			TT_01_01													:= m01_rs1_r1._01_TT_01,
			TT_01_01_offset												:= m01_rs1_r1.cart01_front_temp_offset,
			TT_01_01_error												:= m01_rs1_r1._01_TT_01_Error,
			TT_01_03													:= m01_rs1_r1._01_TT_03,               
			TT_01_03_offset												:= m01_rs1_r1.cart01_front_temp_offset,
			TT_01_03_error												:= m01_rs1_r1._01_TT_03_Error,         
			TT_02_01													:= m01_rs1_r1._02_TT_01,               
			TT_02_01_offset												:= m01_rs1_r1.cart02_front_temp_offset,
			TT_02_01_error												:= m01_rs1_r1._02_TT_01_Error,         
			TT_02_03													:= m01_rs1_r1._02_TT_03,               
			TT_02_03_offset												:= m01_rs1_r1.cart02_front_temp_offset,
			TT_02_03_error												:= m01_rs1_r1._02_TT_03_Error,         
			TT_03_01													:= m01_rs1_r1._03_TT_01,               
			TT_03_01_offset												:= m01_rs1_r1.cart03_front_temp_offset,
			TT_03_01_error												:= m01_rs1_r1._03_TT_01_Error,         
			TT_03_03													:= m01_rs1_r1._03_TT_03,               
			TT_03_03_offset												:= m01_rs1_r1.cart03_front_temp_offset,
			TT_03_03_error												:= m01_rs1_r1._03_TT_03_Error,         
			TT_04_01													:= m01_rs1_r1._04_TT_01,               
			TT_04_01_offset												:= m01_rs1_r1.cart04_front_temp_offset,
			TT_04_01_error												:= m01_rs1_r1._04_TT_01_Error,         
			TT_04_03													:= m01_rs1_r1._04_TT_03,               
			TT_04_03_offset												:= m01_rs1_r1.cart04_front_temp_offset,
			TT_04_03_error												:= m01_rs1_r1._04_TT_03_Error,         
			TT_05_01													:= m01_rs1_r1._05_TT_01,               
			TT_05_01_offset												:= m01_rs1_r1.cart05_front_temp_offset,
			TT_05_01_error												:= m01_rs1_r1._05_TT_01_Error,         
			TT_05_03													:= m01_rs1_r1._05_TT_03,               
			TT_05_03_offset												:= m01_rs1_r1.cart05_front_temp_offset,
			TT_05_03_error												:= m01_rs1_r1._05_TT_03_Error,         
			TT_06_01													:= m01_rs1_r1._06_TT_01,               
			TT_06_01_offset												:= m01_rs1_r1.cart06_front_temp_offset,
			TT_06_01_error												:= m01_rs1_r1._06_TT_01_Error,         
			TT_06_03													:= m01_rs1_r1._06_TT_03,               
			TT_06_03_offset												:= m01_rs1_r1.cart06_front_temp_offset,
			TT_06_03_error												:= m01_rs1_r1._06_TT_03_Error,         
			TT_07_01													:= m01_rs1_r1._07_TT_01,               
			TT_07_01_offset												:= m01_rs1_r1.cart07_front_temp_offset,
			TT_07_01_error												:= m01_rs1_r1._07_TT_01_Error,         
			TT_07_03													:= m01_rs1_r1._07_TT_03,               
			TT_07_03_offset												:= m01_rs1_r1.cart07_front_temp_offset,
			TT_07_03_error												:= m01_rs1_r1._07_TT_03_Error,         
			TT_08_01													:= m01_rs1_r1._08_TT_01,               
			TT_08_01_offset												:= m01_rs1_r1.cart08_front_temp_offset,
			TT_08_01_error												:= m01_rs1_r1._08_TT_01_Error,         
			TT_08_03													:= m01_rs1_r1._08_TT_03,               
			TT_08_03_offset												:= m01_rs1_r1.cart08_front_temp_offset,
			TT_08_03_error												:= m01_rs1_r1._08_TT_03_Error,         
			TT_09_01													:= m01_rs1_r1._09_TT_01,               
			TT_09_01_offset												:= m01_rs1_r1.cart09_front_temp_offset,
			TT_09_01_error												:= m01_rs1_r1._09_TT_01_Error,         
			TT_09_03													:= m01_rs1_r1._09_TT_03,               
			TT_09_03_offset												:= m01_rs1_r1.cart09_front_temp_offset,
			TT_09_03_error												:= m01_rs1_r1._09_TT_03_Error,         
			TT_10_01													:= m01_rs1_r1._10_TT_01,               
			TT_10_01_offset												:= m01_rs1_r1.cart10_front_temp_offset,
			TT_10_01_error												:= m01_rs1_r1._10_TT_01_Error,         
			TT_10_03													:= m01_rs1_r1._10_TT_03,               
			TT_10_03_offset												:= m01_rs1_r1.cart10_front_temp_offset,
			TT_10_03_error												:= m01_rs1_r1._10_TT_03_Error,         
			TT_11_01													:= m01_rs1_r1._11_TT_01,               
			TT_11_01_offset												:= m01_rs1_r1.cart11_front_temp_offset,
			TT_11_01_error												:= m01_rs1_r1._11_TT_01_Error,         
			TT_11_03													:= m01_rs1_r1._11_TT_03,               
			TT_11_03_offset												:= m01_rs1_r1.cart11_front_temp_offset,
			TT_11_03_error												:= m01_rs1_r1._11_TT_03_Error,         
			TT_12_01													:= m01_rs1_r1._12_TT_01,               
			TT_12_01_offset												:= m01_rs1_r1.cart12_front_temp_offset,
			TT_12_01_error												:= m01_rs1_r1._12_TT_01_Error,         
			TT_12_03													:= m01_rs1_r1._12_TT_03,               
			TT_12_03_offset												:= m01_rs1_r1.cart12_front_temp_offset,
			TT_12_03_error												:= m01_rs1_r1._12_TT_03_Error,
			
			cart01_front_temp											=> m01_rs1_r1.cart01_front_temp,						
			cart01_front_temp_error 									=> m01_rs1_r1.cart01_front_temp_error,
			cart01_back_temp											=> m01_rs1_r1.cart01_back_temp,
			cart01_back_temp_error 										=> m01_rs1_r1.cart01_back_temp_error,
			cart02_front_temp											=> m01_rs1_r1.cart02_front_temp,						
			cart02_front_temp_error 									=> m01_rs1_r1.cart02_front_temp_error,
			cart02_back_temp											=> m01_rs1_r1.cart02_back_temp,
			cart02_back_temp_error 										=> m01_rs1_r1.cart02_back_temp_error,
			cart03_front_temp											=> m01_rs1_r1.cart03_front_temp,						
			cart03_front_temp_error 									=> m01_rs1_r1.cart03_front_temp_error,
			cart03_back_temp											=> m01_rs1_r1.cart03_back_temp,
			cart03_back_temp_error 										=> m01_rs1_r1.cart03_back_temp_error,
			cart04_front_temp											=> m01_rs1_r1.cart04_front_temp,						
			cart04_front_temp_error 									=> m01_rs1_r1.cart04_front_temp_error,
			cart04_back_temp											=> m01_rs1_r1.cart04_back_temp,
			cart04_back_temp_error 										=> m01_rs1_r1.cart04_back_temp_error,
			cart05_front_temp											=> m01_rs1_r1.cart05_front_temp,						
			cart05_front_temp_error 									=> m01_rs1_r1.cart05_front_temp_error,
			cart05_back_temp											=> m01_rs1_r1.cart05_back_temp,
			cart05_back_temp_error 										=> m01_rs1_r1.cart05_back_temp_error,
			cart06_front_temp											=> m01_rs1_r1.cart06_front_temp,						
			cart06_front_temp_error 									=> m01_rs1_r1.cart06_front_temp_error,
			cart06_back_temp											=> m01_rs1_r1.cart06_back_temp,
			cart06_back_temp_error 										=> m01_rs1_r1.cart06_back_temp_error,
			cart07_front_temp											=> m01_rs1_r1.cart07_front_temp,						
			cart07_front_temp_error 									=> m01_rs1_r1.cart07_front_temp_error,
			cart07_back_temp											=> m01_rs1_r1.cart07_back_temp,
			cart07_back_temp_error 										=> m01_rs1_r1.cart07_back_temp_error,
			cart08_front_temp											=> m01_rs1_r1.cart08_front_temp,						
			cart08_front_temp_error 									=> m01_rs1_r1.cart08_front_temp_error,
			cart08_back_temp											=> m01_rs1_r1.cart08_back_temp,
			cart08_back_temp_error 										=> m01_rs1_r1.cart08_back_temp_error,
			cart09_front_temp											=> m01_rs1_r1.cart09_front_temp,						
			cart09_front_temp_error 									=> m01_rs1_r1.cart09_front_temp_error,
			cart09_back_temp											=> m01_rs1_r1.cart09_back_temp,
			cart09_back_temp_error 										=> m01_rs1_r1.cart09_back_temp_error,
			cart10_front_temp											=> m01_rs1_r1.cart10_front_temp,						
			cart10_front_temp_error 									=> m01_rs1_r1.cart10_front_temp_error,
			cart10_back_temp											=> m01_rs1_r1.cart10_back_temp,
			cart10_back_temp_error 										=> m01_rs1_r1.cart10_back_temp_error,
			cart11_front_temp											=> m01_rs1_r1.cart11_front_temp,						
			cart11_front_temp_error 									=> m01_rs1_r1.cart11_front_temp_error,
			cart11_back_temp											=> m01_rs1_r1.cart11_back_temp,
			cart11_back_temp_error 										=> m01_rs1_r1.cart11_back_temp_error,
			cart12_front_temp											=> m01_rs1_r1.cart12_front_temp,						
			cart12_front_temp_error 									=> m01_rs1_r1.cart12_front_temp_error,
			cart12_back_temp											=> m01_rs1_r1.cart12_back_temp,
			cart12_back_temp_error 										=> m01_rs1_r1.cart12_back_temp_error,
			         
		                                                        
			inlet_co2_pump												:= m01_rs1_r1.inlet_co2_pump,
			AT_01_pump													=> m01_rs1_r1.AT_01_pump,
			inlet_co2_pump_cmd_status									=> m01_rs1_r1.inlet_co2_pump_cmd_status,
			inlet_co2_sol												:= m01_rs1_r1.inlet_co2_sol,
			AT_01_sol													=> m01_rs1_r1.AT_01_sol,
			inlet_co2_sol_cmd_status									=> m01_rs1_r1.inlet_co2_sol_cmd_status,
			outlet_co2_pump												:= m01_rs1_r1.outlet_co2_pump,
			AT_03_pump													=> m01_rs1_r1.AT_03_pump,
			outlet_co2_pump_cmd_status									=> m01_rs1_r1.outlet_co2_pump_cmd_status,
			outlet_co2_sol												:= m01_rs1_r1.outlet_co2_sol,
			AT_03_sol													=> m01_rs1_r1.AT_03_sol,
			outlet_co2_sol_cmd_status									=> m01_rs1_r1.outlet_co2_sol_cmd_status,
			repres_valve												:= m01_rs1_r1.repres_valve,
			XV_02														=> m01_rs1_r1.XV_02,
			repres_valve_open_cmd_status								=> m01_rs1_r1.repres_valve_open_cmd_status,
			repres_valve_open											:= m01_rs1_r1.repres_valve_open,
			repres_valve_closed											:= m01_rs1_r1.repres_valve_closed,
    	                                                        
			fan_vfd_control												=> m01_rs1_r1.fan_vfd_control,  		
			fan_vfd_target_vel	 		                                => m01_rs1_r1.fan_vfd_target_vel, 
			fan_vfd_enabled	 		                                    => m01_rs1_r1.fan_vfd_enabled, 
			fan_vfd_error		                                        => m01_rs1_r1.fan_vfd_error,
			fan_vfd_output												=> m01_rs1_r1.fan_vfd_output,
			fan_vfd_reset												:= m01_rs1_r1.fan_vfd_reset,
			fan_vfd_enable												:= m01_rs1_r1.fan_vfd_enable,
			fan_vfd_ecat_state											:= m01_rs1_r1.fan_vfd_ecat_state,
			fan_vfd_status												:= m01_rs1_r1.fan_vfd_status,
			fan_vfd														:= m01_rs1_r1.fan_vfd,
			fan_vfd_velocity											:= m01_rs1_r1.fan_vfd_velocity,
			fan_vfd_current												:= m01_rs1_r1.fan_vfd_current,
			fan_vfd_current_amps										=> m01_rs1_r1.fan_vfd_output_current,
			fan_vfd_temp												:= m01_rs1_r1.fan_vfd_temp,
			fan_vfd_temp_degC											=> m01_rs1_r1.fan_vfd_temperature,
			                                                    
			inlet_door_clamps_extend									:= m01_rs1_r1.inlet_door_clamps_extend,
			outlet_door_clamps_extend									:= m01_rs1_r1.outlet_door_clamps_extend,
			inlet_door_clamps_retract									:= m01_rs1_r1.inlet_door_clamps_retract,
			outlet_door_clamps_retract									:= m01_rs1_r1.outlet_door_clamps_retract,
			                                                    
			extend_clamps												:= extend_clamps,
			retract_clamps												:= retract_clamps,
			                                                    
			inlet_door_left_clamps_extend								=> m01_rs1_r1.XV_01_Left_Extend_Solenoid_Valve,
			inlet_door_right_clamps_extend								=> m01_rs1_r1.XV_01_Right_Extend_Solenoid_Valve,
			outlet_door_left_clamps_extend								=> m01_rs1_r1.XV_03_Left_Extend_Solenoid_Valve,
			outlet_door_right_clamps_extend								=> m01_rs1_r1.XV_03_Right_Extend_Solenoid_Valve,
			inlet_door_left_clamps_retract								=> m01_rs1_r1.XV_01_Left_Retract_Solenoid_Valve,
			inlet_door_right_clamps_retract								=> m01_rs1_r1.XV_01_Right_Retract_Solenoid_Valve,
			outlet_door_left_clamps_retract								=> m01_rs1_r1.XV_03_Left_Retract_Solenoid_Valve,
			outlet_door_right_clamps_retract							=> m01_rs1_r1.XV_03_Right_Retract_Solenoid_Valve,
    	                                                        
			inlet_door_left_clamps_extended								:= m01_rs1_r1.inlet_door_left_clamps_extended_ls,  
			inlet_door_right_clamps_extended							:= m01_rs1_r1.inlet_door_right_clamps_extended_ls, 
			outlet_door_left_clamps_extended							:= m01_rs1_r1.outlet_door_left_clamps_extended_ls, 
			outlet_door_right_clamps_extended							:= m01_rs1_r1.outlet_door_right_clamps_extended_ls,
			                                                    
			inlet_door_open												:= m01_rs1_r1.inlet_door_open,
			inlet_door_close											:= m01_rs1_r1.inlet_door_close,
			outlet_door_open											:= m01_rs1_r1.outlet_door_open,
			outlet_door_close											:= m01_rs1_r1.outlet_door_close,
			                                                    
			open_doors													:= open_doors,
			close_doors													:= close_doors,
			                                                    
			open_inlet_door												=> m01_rs1_r1.XV_01_Door_Open_Solenoid_Valve,
			close_inlet_door											=> m01_rs1_r1.XV_01_Door_Close_Solenoid_Valve,
			open_outlet_door											=> m01_rs1_r1.XV_03_Door_Open_Solenoid_Valve,
			close_outlet_door											=> m01_rs1_r1.XV_03_Door_Close_Solenoid_Valve,
			                                                    
			inlet_door_left_open										:= m01_rs1_r1.inlet_door_left_open_ls, 
			inlet_door_right_open										:= m01_rs1_r1.inlet_door_right_open_ls, 
			outlet_door_left_open										:= m01_rs1_r1.outlet_door_left_open_ls, 
			outlet_door_right_open										:= m01_rs1_r1.outlet_door_right_open_ls,
			inlet_door_left_closed										:= m01_rs1_r1.inlet_door_left_closed_ls, 
			inlet_door_right_closed										:= m01_rs1_r1.inlet_door_right_closed_ls, 
			outlet_door_left_closed										:= m01_rs1_r1.outlet_door_left_closed_ls, 
			outlet_door_right_closed									:= m01_rs1_r1.outlet_door_right_closed_ls,
			                                                    
			vacuum_cooling_high_temp_count								=> m01_rs1_r1.vacuum_cooling_high_temp_count,
			adsorption_high_temp_count									=> m01_rs1_r1.adsorption_high_temp_count,
			desorption_high_temp_count									=> m01_rs1_r1.desorption_air_high_temp_count);
END_ACTION

ACTION A_Reactor2_IO:
// Phase 0 - P_M01_RS01.A_Reactor2_IO
// Rev 1.0 - April 26, 2024

fb_R2_IO(	RSet														:= _RS01,
			React														:= _R2,
			
			Power_On													:= m01_rs1.power_control,
			                                                    
			sorbent_low_temp											=> m01_rs1_r2.temp_low,
			sorbent_high_temp											=> m01_rs1_r2.temp_high,
			sorbent_average_temp										=> m01_rs1_r2.temp_average,
			                                                    
			TT_01_01													:= m01_rs1_r2._01_TT_01,
			TT_01_01_offset												:= m01_rs1_r2.cart01_front_temp_offset,
			TT_01_01_error												:= m01_rs1_r2._01_TT_01_Error,
			TT_01_03													:= m01_rs1_r2._01_TT_03,               
			TT_01_03_offset												:= m01_rs1_r2.cart01_front_temp_offset,
			TT_01_03_error												:= m01_rs1_r2._01_TT_03_Error,         
			TT_02_01													:= m01_rs1_r2._02_TT_01,               
			TT_02_01_offset												:= m01_rs1_r2.cart02_front_temp_offset,
			TT_02_01_error												:= m01_rs1_r2._02_TT_01_Error,         
			TT_02_03													:= m01_rs1_r2._02_TT_03,               
			TT_02_03_offset												:= m01_rs1_r2.cart02_front_temp_offset,
			TT_02_03_error												:= m01_rs1_r2._02_TT_03_Error,         
			TT_03_01													:= m01_rs1_r2._03_TT_01,               
			TT_03_01_offset												:= m01_rs1_r2.cart03_front_temp_offset,
			TT_03_01_error												:= m01_rs1_r2._03_TT_01_Error,         
			TT_03_03													:= m01_rs1_r2._03_TT_03,               
			TT_03_03_offset												:= m01_rs1_r2.cart03_front_temp_offset,
			TT_03_03_error												:= m01_rs1_r2._03_TT_03_Error,         
			TT_04_01													:= m01_rs1_r2._04_TT_01,               
			TT_04_01_offset												:= m01_rs1_r2.cart04_front_temp_offset,
			TT_04_01_error												:= m01_rs1_r2._04_TT_01_Error,         
			TT_04_03													:= m01_rs1_r2._04_TT_03,               
			TT_04_03_offset												:= m01_rs1_r2.cart04_front_temp_offset,
			TT_04_03_error												:= m01_rs1_r2._04_TT_03_Error,         
			TT_05_01													:= m01_rs1_r2._05_TT_01,               
			TT_05_01_offset												:= m01_rs1_r2.cart05_front_temp_offset,
			TT_05_01_error												:= m01_rs1_r2._05_TT_01_Error,         
			TT_05_03													:= m01_rs1_r2._05_TT_03,               
			TT_05_03_offset												:= m01_rs1_r2.cart05_front_temp_offset,
			TT_05_03_error												:= m01_rs1_r2._05_TT_03_Error,         
			TT_06_01													:= m01_rs1_r2._06_TT_01,               
			TT_06_01_offset												:= m01_rs1_r2.cart06_front_temp_offset,
			TT_06_01_error												:= m01_rs1_r2._06_TT_01_Error,         
			TT_06_03													:= m01_rs1_r2._06_TT_03,               
			TT_06_03_offset												:= m01_rs1_r2.cart06_front_temp_offset,
			TT_06_03_error												:= m01_rs1_r2._06_TT_03_Error,         
			TT_07_01													:= m01_rs1_r2._07_TT_01,               
			TT_07_01_offset												:= m01_rs1_r2.cart07_front_temp_offset,
			TT_07_01_error												:= m01_rs1_r2._07_TT_01_Error,         
			TT_07_03													:= m01_rs1_r2._07_TT_03,               
			TT_07_03_offset												:= m01_rs1_r2.cart07_front_temp_offset,
			TT_07_03_error												:= m01_rs1_r2._07_TT_03_Error,         
			TT_08_01													:= m01_rs1_r2._08_TT_01,               
			TT_08_01_offset												:= m01_rs1_r2.cart08_front_temp_offset,
			TT_08_01_error												:= m01_rs1_r2._08_TT_01_Error,         
			TT_08_03													:= m01_rs1_r2._08_TT_03,               
			TT_08_03_offset												:= m01_rs1_r2.cart08_front_temp_offset,
			TT_08_03_error												:= m01_rs1_r2._08_TT_03_Error,         
			TT_09_01													:= m01_rs1_r2._09_TT_01,               
			TT_09_01_offset												:= m01_rs1_r2.cart09_front_temp_offset,
			TT_09_01_error												:= m01_rs1_r2._09_TT_01_Error,         
			TT_09_03													:= m01_rs1_r2._09_TT_03,               
			TT_09_03_offset												:= m01_rs1_r2.cart09_front_temp_offset,
			TT_09_03_error												:= m01_rs1_r2._09_TT_03_Error,         
			TT_10_01													:= m01_rs1_r2._10_TT_01,               
			TT_10_01_offset												:= m01_rs1_r2.cart10_front_temp_offset,
			TT_10_01_error												:= m01_rs1_r2._10_TT_01_Error,         
			TT_10_03													:= m01_rs1_r2._10_TT_03,               
			TT_10_03_offset												:= m01_rs1_r2.cart10_front_temp_offset,
			TT_10_03_error												:= m01_rs1_r2._10_TT_03_Error,         
			TT_11_01													:= m01_rs1_r2._11_TT_01,               
			TT_11_01_offset												:= m01_rs1_r2.cart11_front_temp_offset,
			TT_11_01_error												:= m01_rs1_r2._11_TT_01_Error,         
			TT_11_03													:= m01_rs1_r2._11_TT_03,               
			TT_11_03_offset												:= m01_rs1_r2.cart11_front_temp_offset,
			TT_11_03_error												:= m01_rs1_r2._11_TT_03_Error,         
			TT_12_01													:= m01_rs1_r2._12_TT_01,               
			TT_12_01_offset												:= m01_rs1_r2.cart12_front_temp_offset,
			TT_12_01_error												:= m01_rs1_r2._12_TT_01_Error,         
			TT_12_03													:= m01_rs1_r2._12_TT_03,               
			TT_12_03_offset												:= m01_rs1_r2.cart12_front_temp_offset,
			TT_12_03_error												:= m01_rs1_r2._12_TT_03_Error,  

			cart01_front_temp											=> m01_rs1_r2.cart01_front_temp,						
			cart01_front_temp_error 									=> m01_rs1_r2.cart01_front_temp_error,
			cart01_back_temp											=> m01_rs1_r2.cart01_back_temp,
			cart01_back_temp_error 										=> m01_rs1_r2.cart01_back_temp_error,
			cart02_front_temp											=> m01_rs1_r2.cart02_front_temp,						
			cart02_front_temp_error 									=> m01_rs1_r2.cart02_front_temp_error,
			cart02_back_temp											=> m01_rs1_r2.cart02_back_temp,
			cart02_back_temp_error 										=> m01_rs1_r2.cart02_back_temp_error,
			cart03_front_temp											=> m01_rs1_r2.cart03_front_temp,						
			cart03_front_temp_error 									=> m01_rs1_r2.cart03_front_temp_error,
			cart03_back_temp											=> m01_rs1_r2.cart03_back_temp,
			cart03_back_temp_error 										=> m01_rs1_r2.cart03_back_temp_error,
			cart04_front_temp											=> m01_rs1_r2.cart04_front_temp,						
			cart04_front_temp_error 									=> m01_rs1_r2.cart04_front_temp_error,
			cart04_back_temp											=> m01_rs1_r2.cart04_back_temp,
			cart04_back_temp_error 										=> m01_rs1_r2.cart04_back_temp_error,
			cart05_front_temp											=> m01_rs1_r2.cart05_front_temp,						
			cart05_front_temp_error 									=> m01_rs1_r2.cart05_front_temp_error,
			cart05_back_temp											=> m01_rs1_r2.cart05_back_temp,
			cart05_back_temp_error 										=> m01_rs1_r2.cart05_back_temp_error,
			cart06_front_temp											=> m01_rs1_r2.cart06_front_temp,						
			cart06_front_temp_error 									=> m01_rs1_r2.cart06_front_temp_error,
			cart06_back_temp											=> m01_rs1_r2.cart06_back_temp,
			cart06_back_temp_error 										=> m01_rs1_r2.cart06_back_temp_error,
			cart07_front_temp											=> m01_rs1_r2.cart07_front_temp,						
			cart07_front_temp_error 									=> m01_rs1_r2.cart07_front_temp_error,
			cart07_back_temp											=> m01_rs1_r2.cart07_back_temp,
			cart07_back_temp_error 										=> m01_rs1_r2.cart07_back_temp_error,
			cart08_front_temp											=> m01_rs1_r2.cart08_front_temp,						
			cart08_front_temp_error 									=> m01_rs1_r2.cart08_front_temp_error,
			cart08_back_temp											=> m01_rs1_r2.cart08_back_temp,
			cart08_back_temp_error 										=> m01_rs1_r2.cart08_back_temp_error,
			cart09_front_temp											=> m01_rs1_r2.cart09_front_temp,						
			cart09_front_temp_error 									=> m01_rs1_r2.cart09_front_temp_error,
			cart09_back_temp											=> m01_rs1_r2.cart09_back_temp,
			cart09_back_temp_error 										=> m01_rs1_r2.cart09_back_temp_error,
			cart10_front_temp											=> m01_rs1_r2.cart10_front_temp,						
			cart10_front_temp_error 									=> m01_rs1_r2.cart10_front_temp_error,
			cart10_back_temp											=> m01_rs1_r2.cart10_back_temp,
			cart10_back_temp_error 										=> m01_rs1_r2.cart10_back_temp_error,
			cart11_front_temp											=> m01_rs1_r2.cart11_front_temp,						
			cart11_front_temp_error 									=> m01_rs1_r2.cart11_front_temp_error,
			cart11_back_temp											=> m01_rs1_r2.cart11_back_temp,
			cart11_back_temp_error 										=> m01_rs1_r2.cart11_back_temp_error,
			cart12_front_temp											=> m01_rs1_r2.cart12_front_temp,						
			cart12_front_temp_error 									=> m01_rs1_r2.cart12_front_temp_error,
			cart12_back_temp											=> m01_rs1_r2.cart12_back_temp,
			cart12_back_temp_error 										=> m01_rs1_r2.cart12_back_temp_error,       
		                                                        
			inlet_co2_pump												:= m01_rs1_r2.inlet_co2_pump,
			AT_01_pump													=> m01_rs1_r2.AT_01_pump,
			inlet_co2_pump_cmd_status									=> m01_rs1_r2.inlet_co2_pump_cmd_status,
			inlet_co2_sol												:= m01_rs1_r2.inlet_co2_sol,
			AT_01_sol													=> m01_rs1_r2.AT_01_sol,
			inlet_co2_sol_cmd_status									=> m01_rs1_r2.inlet_co2_sol_cmd_status,
			outlet_co2_pump												:= m01_rs1_r2.outlet_co2_pump,
			AT_03_pump													=> m01_rs1_r2.AT_03_pump,
			outlet_co2_pump_cmd_status									=> m01_rs1_r2.outlet_co2_pump_cmd_status,
			outlet_co2_sol												:= m01_rs1_r2.outlet_co2_sol,
			AT_03_sol													=> m01_rs1_r2.AT_03_sol,
			outlet_co2_sol_cmd_status									=> m01_rs1_r2.outlet_co2_sol_cmd_status,
			repres_valve												:= m01_rs1_r2.repres_valve,
			XV_02														=> m01_rs1_r2.XV_02,
			repres_valve_open_cmd_status								=> m01_rs1_r2.repres_valve_open_cmd_status,
			repres_valve_open											:= m01_rs1_r2.repres_valve_open,
			repres_valve_closed											:= m01_rs1_r2.repres_valve_closed,
    	                                                        
			fan_vfd_control												=> m01_rs1_r2.fan_vfd_control,  		
			fan_vfd_target_vel	 		                                => m01_rs1_r2.fan_vfd_target_vel, 
			fan_vfd_enabled	 		                                    => m01_rs1_r2.fan_vfd_enabled, 
			fan_vfd_error		                                        => m01_rs1_r2.fan_vfd_error,
			fan_vfd_output												=> m01_rs1_r2.fan_vfd_output,
			fan_vfd_reset												:= m01_rs1_r2.fan_vfd_reset,
			fan_vfd_enable												:= m01_rs1_r2.fan_vfd_enable,
			fan_vfd_ecat_state											:= m01_rs1_r2.fan_vfd_ecat_state,
			fan_vfd_status												:= m01_rs1_r2.fan_vfd_status,
			fan_vfd														:= m01_rs1_r2.fan_vfd,
			fan_vfd_velocity											:= m01_rs1_r2.fan_vfd_velocity,
			fan_vfd_current												:= m01_rs1_r2.fan_vfd_current,
			fan_vfd_current_amps										=> m01_rs1_r2.fan_vfd_output_current,
			                                                    
			inlet_door_clamps_extend									:= m01_rs1_r2.inlet_door_clamps_extend,
			outlet_door_clamps_extend									:= m01_rs1_r2.outlet_door_clamps_extend,
			inlet_door_clamps_retract									:= m01_rs1_r2.inlet_door_clamps_retract,
			outlet_door_clamps_retract									:= m01_rs1_r2.outlet_door_clamps_retract,
			                                                    
			extend_clamps												:= extend_clamps,
			retract_clamps												:= retract_clamps,
			                                                    
			inlet_door_left_clamps_extend								=> m01_rs1_r2.XV_01_Left_Extend_Solenoid_Valve,
			inlet_door_right_clamps_extend								=> m01_rs1_r2.XV_01_Right_Extend_Solenoid_Valve,
			outlet_door_left_clamps_extend								=> m01_rs1_r2.XV_03_Left_Extend_Solenoid_Valve,
			outlet_door_right_clamps_extend								=> m01_rs1_r2.XV_03_Right_Extend_Solenoid_Valve,
			inlet_door_left_clamps_retract								=> m01_rs1_r2.XV_01_Left_Retract_Solenoid_Valve,
			inlet_door_right_clamps_retract								=> m01_rs1_r2.XV_01_Right_Retract_Solenoid_Valve,
			outlet_door_left_clamps_retract								=> m01_rs1_r2.XV_03_Left_Retract_Solenoid_Valve,
			outlet_door_right_clamps_retract							=> m01_rs1_r2.XV_03_Right_Retract_Solenoid_Valve,
    	                                                        
			inlet_door_left_clamps_extended								:= m01_rs1_r2.inlet_door_left_clamps_extended_ls,  
			inlet_door_right_clamps_extended							:= m01_rs1_r2.inlet_door_right_clamps_extended_ls, 
			outlet_door_left_clamps_extended							:= m01_rs1_r2.outlet_door_left_clamps_extended_ls, 
			outlet_door_right_clamps_extended							:= m01_rs1_r2.outlet_door_right_clamps_extended_ls,
			                                                    
			inlet_door_open												:= m01_rs1_r2.inlet_door_open,
			inlet_door_close											:= m01_rs1_r2.inlet_door_close,
			outlet_door_open											:= m01_rs1_r2.outlet_door_open,
			outlet_door_close											:= m01_rs1_r2.outlet_door_close,
			                                                    
			open_doors													:= open_doors,
			close_doors													:= close_doors,
			                                                    
			open_inlet_door												=> m01_rs1_r2.XV_01_Door_Open_Solenoid_Valve,
			close_inlet_door											=> m01_rs1_r2.XV_01_Door_Close_Solenoid_Valve,
			open_outlet_door											=> m01_rs1_r2.XV_03_Door_Open_Solenoid_Valve,
			close_outlet_door											=> m01_rs1_r2.XV_03_Door_Close_Solenoid_Valve,
			                                                    
			inlet_door_left_open										:= m01_rs1_r2.inlet_door_left_open_ls, 
			inlet_door_right_open										:= m01_rs1_r2.inlet_door_right_open_ls, 
			outlet_door_left_open										:= m01_rs1_r2.outlet_door_left_open_ls, 
			outlet_door_right_open										:= m01_rs1_r2.outlet_door_right_open_ls,
			inlet_door_left_closed										:= m01_rs1_r2.inlet_door_left_closed_ls, 
			inlet_door_right_closed										:= m01_rs1_r2.inlet_door_right_closed_ls, 
			outlet_door_left_closed										:= m01_rs1_r2.outlet_door_left_closed_ls, 
			outlet_door_right_closed									:= m01_rs1_r2.outlet_door_right_closed_ls,
			                                                    
			vacuum_cooling_high_temp_count								=> m01_rs1_r2.vacuum_cooling_high_temp_count,
			adsorption_high_temp_count									=> m01_rs1_r2.adsorption_high_temp_count,
			desorption_high_temp_count									=> m01_rs1_r2.desorption_air_high_temp_count);
END_ACTION

ACTION A_Reactor3_IO:
// Phase 0 - P_M01_RS01.A_Reactor3_IO
// Rev 1.0 - April 26, 2024

fb_R3_IO(	RSet														:= _RS01,
			React														:= _R3,
			
			Power_On													:= m01_rs1.power_control,
			                                                    
			sorbent_low_temp											=> m01_rs1_r3.temp_low,
			sorbent_high_temp											=> m01_rs1_r3.temp_high,
			sorbent_average_temp										=> m01_rs1_r3.temp_average,
			                                                    
			TT_01_01													:= m01_rs1_r3._01_TT_01,
			TT_01_01_offset												:= m01_rs1_r3.cart01_front_temp_offset,
			TT_01_01_error												:= m01_rs1_r3._01_TT_01_Error,
			TT_01_03													:= m01_rs1_r3._01_TT_03,               
			TT_01_03_offset												:= m01_rs1_r3.cart01_front_temp_offset,
			TT_01_03_error												:= m01_rs1_r3._01_TT_03_Error,         
			TT_02_01													:= m01_rs1_r3._02_TT_01,               
			TT_02_01_offset												:= m01_rs1_r3.cart02_front_temp_offset,
			TT_02_01_error												:= m01_rs1_r3._02_TT_01_Error,         
			TT_02_03													:= m01_rs1_r3._02_TT_03,               
			TT_02_03_offset												:= m01_rs1_r3.cart02_front_temp_offset,
			TT_02_03_error												:= m01_rs1_r3._02_TT_03_Error,         
			TT_03_01													:= m01_rs1_r3._03_TT_01,               
			TT_03_01_offset												:= m01_rs1_r3.cart03_front_temp_offset,
			TT_03_01_error												:= m01_rs1_r3._03_TT_01_Error,         
			TT_03_03													:= m01_rs1_r3._03_TT_03,               
			TT_03_03_offset												:= m01_rs1_r3.cart03_front_temp_offset,
			TT_03_03_error												:= m01_rs1_r3._03_TT_03_Error,         
			TT_04_01													:= m01_rs1_r3._04_TT_01,               
			TT_04_01_offset												:= m01_rs1_r3.cart04_front_temp_offset,
			TT_04_01_error												:= m01_rs1_r3._04_TT_01_Error,         
			TT_04_03													:= m01_rs1_r3._04_TT_03,               
			TT_04_03_offset												:= m01_rs1_r3.cart04_front_temp_offset,
			TT_04_03_error												:= m01_rs1_r3._04_TT_03_Error,         
			TT_05_01													:= m01_rs1_r3._05_TT_01,               
			TT_05_01_offset												:= m01_rs1_r3.cart05_front_temp_offset,
			TT_05_01_error												:= m01_rs1_r3._05_TT_01_Error,         
			TT_05_03													:= m01_rs1_r3._05_TT_03,               
			TT_05_03_offset												:= m01_rs1_r3.cart05_front_temp_offset,
			TT_05_03_error												:= m01_rs1_r3._05_TT_03_Error,         
			TT_06_01													:= m01_rs1_r3._06_TT_01,               
			TT_06_01_offset												:= m01_rs1_r3.cart06_front_temp_offset,
			TT_06_01_error												:= m01_rs1_r3._06_TT_01_Error,         
			TT_06_03													:= m01_rs1_r3._06_TT_03,               
			TT_06_03_offset												:= m01_rs1_r3.cart06_front_temp_offset,
			TT_06_03_error												:= m01_rs1_r3._06_TT_03_Error,         
			TT_07_01													:= m01_rs1_r3._07_TT_01,               
			TT_07_01_offset												:= m01_rs1_r3.cart07_front_temp_offset,
			TT_07_01_error												:= m01_rs1_r3._07_TT_01_Error,         
			TT_07_03													:= m01_rs1_r3._07_TT_03,               
			TT_07_03_offset												:= m01_rs1_r3.cart07_front_temp_offset,
			TT_07_03_error												:= m01_rs1_r3._07_TT_03_Error,         
			TT_08_01													:= m01_rs1_r3._08_TT_01,               
			TT_08_01_offset												:= m01_rs1_r3.cart08_front_temp_offset,
			TT_08_01_error												:= m01_rs1_r3._08_TT_01_Error,         
			TT_08_03													:= m01_rs1_r3._08_TT_03,               
			TT_08_03_offset												:= m01_rs1_r3.cart08_front_temp_offset,
			TT_08_03_error												:= m01_rs1_r3._08_TT_03_Error,         
			TT_09_01													:= m01_rs1_r3._09_TT_01,               
			TT_09_01_offset												:= m01_rs1_r3.cart09_front_temp_offset,
			TT_09_01_error												:= m01_rs1_r3._09_TT_01_Error,         
			TT_09_03													:= m01_rs1_r3._09_TT_03,               
			TT_09_03_offset												:= m01_rs1_r3.cart09_front_temp_offset,
			TT_09_03_error												:= m01_rs1_r3._09_TT_03_Error,         
			TT_10_01													:= m01_rs1_r3._10_TT_01,               
			TT_10_01_offset												:= m01_rs1_r3.cart10_front_temp_offset,
			TT_10_01_error												:= m01_rs1_r3._10_TT_01_Error,         
			TT_10_03													:= m01_rs1_r3._10_TT_03,               
			TT_10_03_offset												:= m01_rs1_r3.cart10_front_temp_offset,
			TT_10_03_error												:= m01_rs1_r3._10_TT_03_Error,         
			TT_11_01													:= m01_rs1_r3._11_TT_01,               
			TT_11_01_offset												:= m01_rs1_r3.cart11_front_temp_offset,
			TT_11_01_error												:= m01_rs1_r3._11_TT_01_Error,         
			TT_11_03													:= m01_rs1_r3._11_TT_03,               
			TT_11_03_offset												:= m01_rs1_r3.cart11_front_temp_offset,
			TT_11_03_error												:= m01_rs1_r3._11_TT_03_Error,         
			TT_12_01													:= m01_rs1_r3._12_TT_01,               
			TT_12_01_offset												:= m01_rs1_r3.cart12_front_temp_offset,
			TT_12_01_error												:= m01_rs1_r3._12_TT_01_Error,         
			TT_12_03													:= m01_rs1_r3._12_TT_03,               
			TT_12_03_offset												:= m01_rs1_r3.cart12_front_temp_offset,
			TT_12_03_error												:= m01_rs1_r3._12_TT_03_Error, 

			cart01_front_temp											=> m01_rs1_r3.cart01_front_temp,						
			cart01_front_temp_error 									=> m01_rs1_r3.cart01_front_temp_error,
			cart01_back_temp											=> m01_rs1_r3.cart01_back_temp,
			cart01_back_temp_error 										=> m01_rs1_r3.cart01_back_temp_error,
			cart02_front_temp											=> m01_rs1_r3.cart02_front_temp,						
			cart02_front_temp_error 									=> m01_rs1_r3.cart02_front_temp_error,
			cart02_back_temp											=> m01_rs1_r3.cart02_back_temp,
			cart02_back_temp_error 										=> m01_rs1_r3.cart02_back_temp_error,
			cart03_front_temp											=> m01_rs1_r3.cart03_front_temp,						
			cart03_front_temp_error 									=> m01_rs1_r3.cart03_front_temp_error,
			cart03_back_temp											=> m01_rs1_r3.cart03_back_temp,
			cart03_back_temp_error 										=> m01_rs1_r3.cart03_back_temp_error,
			cart04_front_temp											=> m01_rs1_r3.cart04_front_temp,						
			cart04_front_temp_error 									=> m01_rs1_r3.cart04_front_temp_error,
			cart04_back_temp											=> m01_rs1_r3.cart04_back_temp,
			cart04_back_temp_error 										=> m01_rs1_r3.cart04_back_temp_error,
			cart05_front_temp											=> m01_rs1_r3.cart05_front_temp,						
			cart05_front_temp_error 									=> m01_rs1_r3.cart05_front_temp_error,
			cart05_back_temp											=> m01_rs1_r3.cart05_back_temp,
			cart05_back_temp_error 										=> m01_rs1_r3.cart05_back_temp_error,
			cart06_front_temp											=> m01_rs1_r3.cart06_front_temp,						
			cart06_front_temp_error 									=> m01_rs1_r3.cart06_front_temp_error,
			cart06_back_temp											=> m01_rs1_r3.cart06_back_temp,
			cart06_back_temp_error 										=> m01_rs1_r3.cart06_back_temp_error,
			cart07_front_temp											=> m01_rs1_r3.cart07_front_temp,						
			cart07_front_temp_error 									=> m01_rs1_r3.cart07_front_temp_error,
			cart07_back_temp											=> m01_rs1_r3.cart07_back_temp,
			cart07_back_temp_error 										=> m01_rs1_r3.cart07_back_temp_error,
			cart08_front_temp											=> m01_rs1_r3.cart08_front_temp,						
			cart08_front_temp_error 									=> m01_rs1_r3.cart08_front_temp_error,
			cart08_back_temp											=> m01_rs1_r3.cart08_back_temp,
			cart08_back_temp_error 										=> m01_rs1_r3.cart08_back_temp_error,
			cart09_front_temp											=> m01_rs1_r3.cart09_front_temp,						
			cart09_front_temp_error 									=> m01_rs1_r3.cart09_front_temp_error,
			cart09_back_temp											=> m01_rs1_r3.cart09_back_temp,
			cart09_back_temp_error 										=> m01_rs1_r3.cart09_back_temp_error,
			cart10_front_temp											=> m01_rs1_r3.cart10_front_temp,						
			cart10_front_temp_error 									=> m01_rs1_r3.cart10_front_temp_error,
			cart10_back_temp											=> m01_rs1_r3.cart10_back_temp,
			cart10_back_temp_error 										=> m01_rs1_r3.cart10_back_temp_error,
			cart11_front_temp											=> m01_rs1_r3.cart11_front_temp,						
			cart11_front_temp_error 									=> m01_rs1_r3.cart11_front_temp_error,
			cart11_back_temp											=> m01_rs1_r3.cart11_back_temp,
			cart11_back_temp_error 										=> m01_rs1_r3.cart11_back_temp_error,
			cart12_front_temp											=> m01_rs1_r3.cart12_front_temp,						
			cart12_front_temp_error 									=> m01_rs1_r3.cart12_front_temp_error,
			cart12_back_temp											=> m01_rs1_r3.cart12_back_temp,
			cart12_back_temp_error 										=> m01_rs1_r3.cart12_back_temp_error,        
		                                                        
			inlet_co2_pump												:= m01_rs1_r3.inlet_co2_pump,
			AT_01_pump													=> m01_rs1_r3.AT_01_pump,
			inlet_co2_pump_cmd_status									=> m01_rs1_r3.inlet_co2_pump_cmd_status,
			inlet_co2_sol												:= m01_rs1_r3.inlet_co2_sol,
			AT_01_sol													=> m01_rs1_r3.AT_01_sol,
			inlet_co2_sol_cmd_status									=> m01_rs1_r3.inlet_co2_sol_cmd_status,
			outlet_co2_pump												:= m01_rs1_r3.outlet_co2_pump,
			AT_03_pump													=> m01_rs1_r3.AT_03_pump,
			outlet_co2_pump_cmd_status									=> m01_rs1_r3.outlet_co2_pump_cmd_status,
			outlet_co2_sol												:= m01_rs1_r3.outlet_co2_sol,
			AT_03_sol													=> m01_rs1_r3.AT_03_sol,
			outlet_co2_sol_cmd_status									=> m01_rs1_r3.outlet_co2_sol_cmd_status,
			repres_valve												:= m01_rs1_r3.repres_valve,
			XV_02														=> m01_rs1_r3.XV_02,
			repres_valve_open_cmd_status								=> m01_rs1_r3.repres_valve_open_cmd_status,
			repres_valve_open											:= m01_rs1_r3.repres_valve_open,
			repres_valve_closed											:= m01_rs1_r3.repres_valve_closed,
    	                                                        
			fan_vfd_control												=> m01_rs1_r3.fan_vfd_control,  		
			fan_vfd_target_vel	 		                                => m01_rs1_r3.fan_vfd_target_vel, 
			fan_vfd_enabled	 		                                    => m01_rs1_r3.fan_vfd_enabled, 
			fan_vfd_error		                                        => m01_rs1_r3.fan_vfd_error,
			fan_vfd_output												=> m01_rs1_r3.fan_vfd_output,
			fan_vfd_reset												:= m01_rs1_r3.fan_vfd_reset,
			fan_vfd_enable												:= m01_rs1_r3.fan_vfd_enable,
			fan_vfd_ecat_state											:= m01_rs1_r3.fan_vfd_ecat_state,
			fan_vfd_status												:= m01_rs1_r3.fan_vfd_status,
			fan_vfd														:= m01_rs1_r3.fan_vfd,
			fan_vfd_velocity											:= m01_rs1_r3.fan_vfd_velocity,
			fan_vfd_current												:= m01_rs1_r3.fan_vfd_current,
			fan_vfd_current_amps										=> m01_rs1_r3.fan_vfd_output_current,
			                                                    
			inlet_door_clamps_extend									:= m01_rs1_r3.inlet_door_clamps_extend,
			outlet_door_clamps_extend									:= m01_rs1_r3.outlet_door_clamps_extend,
			inlet_door_clamps_retract									:= m01_rs1_r3.inlet_door_clamps_retract,
			outlet_door_clamps_retract									:= m01_rs1_r3.outlet_door_clamps_retract,
			                                                    
			extend_clamps												:= extend_clamps,
			retract_clamps												:= retract_clamps,
			                                                    
			inlet_door_left_clamps_extend								=> m01_rs1_r3.XV_01_Left_Extend_Solenoid_Valve,
			inlet_door_right_clamps_extend								=> m01_rs1_r3.XV_01_Right_Extend_Solenoid_Valve,
			outlet_door_left_clamps_extend								=> m01_rs1_r3.XV_03_Left_Extend_Solenoid_Valve,
			outlet_door_right_clamps_extend								=> m01_rs1_r3.XV_03_Right_Extend_Solenoid_Valve,
			inlet_door_left_clamps_retract								=> m01_rs1_r3.XV_01_Left_Retract_Solenoid_Valve,
			inlet_door_right_clamps_retract								=> m01_rs1_r3.XV_01_Right_Retract_Solenoid_Valve,
			outlet_door_left_clamps_retract								=> m01_rs1_r3.XV_03_Left_Retract_Solenoid_Valve,
			outlet_door_right_clamps_retract							=> m01_rs1_r3.XV_03_Right_Retract_Solenoid_Valve,
    	                                                        
			inlet_door_left_clamps_extended								:= m01_rs1_r3.inlet_door_left_clamps_extended_ls,  
			inlet_door_right_clamps_extended							:= m01_rs1_r3.inlet_door_right_clamps_extended_ls, 
			outlet_door_left_clamps_extended							:= m01_rs1_r3.outlet_door_left_clamps_extended_ls, 
			outlet_door_right_clamps_extended							:= m01_rs1_r3.outlet_door_right_clamps_extended_ls,
			                                                    
			inlet_door_open												:= m01_rs1_r3.inlet_door_open,
			inlet_door_close											:= m01_rs1_r3.inlet_door_close,
			outlet_door_open											:= m01_rs1_r3.outlet_door_open,
			outlet_door_close											:= m01_rs1_r3.outlet_door_close,
			                                                    
			open_doors													:= open_doors,
			close_doors													:= close_doors,
			                                                    
			open_inlet_door												=> m01_rs1_r3.XV_01_Door_Open_Solenoid_Valve,
			close_inlet_door											=> m01_rs1_r3.XV_01_Door_Close_Solenoid_Valve,
			open_outlet_door											=> m01_rs1_r3.XV_03_Door_Open_Solenoid_Valve,
			close_outlet_door											=> m01_rs1_r3.XV_03_Door_Close_Solenoid_Valve,
			                                                    
			inlet_door_left_open										:= m01_rs1_r3.inlet_door_left_open_ls, 
			inlet_door_right_open										:= m01_rs1_r3.inlet_door_right_open_ls, 
			outlet_door_left_open										:= m01_rs1_r3.outlet_door_left_open_ls, 
			outlet_door_right_open										:= m01_rs1_r3.outlet_door_right_open_ls,
			inlet_door_left_closed										:= m01_rs1_r3.inlet_door_left_closed_ls, 
			inlet_door_right_closed										:= m01_rs1_r3.inlet_door_right_closed_ls, 
			outlet_door_left_closed										:= m01_rs1_r3.outlet_door_left_closed_ls, 
			outlet_door_right_closed									:= m01_rs1_r3.outlet_door_right_closed_ls,
			                                                    
			vacuum_cooling_high_temp_count								=> m01_rs1_r3.vacuum_cooling_high_temp_count,
			adsorption_high_temp_count									=> m01_rs1_r3.adsorption_high_temp_count,
			desorption_high_temp_count									=> m01_rs1_r3.desorption_air_high_temp_count);
END_ACTION

ACTION A_Reactor4_IO:
// Phase 0 - P_M01_RS01.A_Reactor4_IO
// Rev 1.0 - April 26, 2024

fb_R4_IO(	RSet														:= _RS01,
			React														:= _R4,
			
			Power_On													:= m01_rs1.power_control,
			                                                    
			sorbent_low_temp											=> m01_rs1_r4.temp_low,
			sorbent_high_temp											=> m01_rs1_r4.temp_high,
			sorbent_average_temp										=> m01_rs1_r4.temp_average,
			                                                    
			TT_01_01													:= m01_rs1_r4._01_TT_01,
			TT_01_01_offset												:= m01_rs1_r4.cart01_front_temp_offset,
			TT_01_01_error												:= m01_rs1_r4._01_TT_01_Error,
			TT_01_03													:= m01_rs1_r4._01_TT_03,               
			TT_01_03_offset												:= m01_rs1_r4.cart01_front_temp_offset,
			TT_01_03_error												:= m01_rs1_r4._01_TT_03_Error,         
			TT_02_01													:= m01_rs1_r4._02_TT_01,               
			TT_02_01_offset												:= m01_rs1_r4.cart02_front_temp_offset,
			TT_02_01_error												:= m01_rs1_r4._02_TT_01_Error,         
			TT_02_03													:= m01_rs1_r4._02_TT_03,               
			TT_02_03_offset												:= m01_rs1_r4.cart02_front_temp_offset,
			TT_02_03_error												:= m01_rs1_r4._02_TT_03_Error,         
			TT_03_01													:= m01_rs1_r4._03_TT_01,               
			TT_03_01_offset												:= m01_rs1_r4.cart03_front_temp_offset,
			TT_03_01_error												:= m01_rs1_r4._03_TT_01_Error,         
			TT_03_03													:= m01_rs1_r4._03_TT_03,               
			TT_03_03_offset												:= m01_rs1_r4.cart03_front_temp_offset,
			TT_03_03_error												:= m01_rs1_r4._03_TT_03_Error,         
			TT_04_01													:= m01_rs1_r4._04_TT_01,               
			TT_04_01_offset												:= m01_rs1_r4.cart04_front_temp_offset,
			TT_04_01_error												:= m01_rs1_r4._04_TT_01_Error,         
			TT_04_03													:= m01_rs1_r4._04_TT_03,               
			TT_04_03_offset												:= m01_rs1_r4.cart04_front_temp_offset,
			TT_04_03_error												:= m01_rs1_r4._04_TT_03_Error,         
			TT_05_01													:= m01_rs1_r4._05_TT_01,               
			TT_05_01_offset												:= m01_rs1_r4.cart05_front_temp_offset,
			TT_05_01_error												:= m01_rs1_r4._05_TT_01_Error,         
			TT_05_03													:= m01_rs1_r4._05_TT_03,               
			TT_05_03_offset												:= m01_rs1_r4.cart05_front_temp_offset,
			TT_05_03_error												:= m01_rs1_r4._05_TT_03_Error,         
			TT_06_01													:= m01_rs1_r4._06_TT_01,               
			TT_06_01_offset												:= m01_rs1_r4.cart06_front_temp_offset,
			TT_06_01_error												:= m01_rs1_r4._06_TT_01_Error,         
			TT_06_03													:= m01_rs1_r4._06_TT_03,               
			TT_06_03_offset												:= m01_rs1_r4.cart06_front_temp_offset,
			TT_06_03_error												:= m01_rs1_r4._06_TT_03_Error,         
			TT_07_01													:= m01_rs1_r4._07_TT_01,               
			TT_07_01_offset												:= m01_rs1_r4.cart07_front_temp_offset,
			TT_07_01_error												:= m01_rs1_r4._07_TT_01_Error,         
			TT_07_03													:= m01_rs1_r4._07_TT_03,               
			TT_07_03_offset												:= m01_rs1_r4.cart07_front_temp_offset,
			TT_07_03_error												:= m01_rs1_r4._07_TT_03_Error,         
			TT_08_01													:= m01_rs1_r4._08_TT_01,               
			TT_08_01_offset												:= m01_rs1_r4.cart08_front_temp_offset,
			TT_08_01_error												:= m01_rs1_r4._08_TT_01_Error,         
			TT_08_03													:= m01_rs1_r4._08_TT_03,               
			TT_08_03_offset												:= m01_rs1_r4.cart08_front_temp_offset,
			TT_08_03_error												:= m01_rs1_r4._08_TT_03_Error,         
			TT_09_01													:= m01_rs1_r4._09_TT_01,               
			TT_09_01_offset												:= m01_rs1_r4.cart09_front_temp_offset,
			TT_09_01_error												:= m01_rs1_r4._09_TT_01_Error,         
			TT_09_03													:= m01_rs1_r4._09_TT_03,               
			TT_09_03_offset												:= m01_rs1_r4.cart09_front_temp_offset,
			TT_09_03_error												:= m01_rs1_r4._09_TT_03_Error,         
			TT_10_01													:= m01_rs1_r4._10_TT_01,               
			TT_10_01_offset												:= m01_rs1_r4.cart10_front_temp_offset,
			TT_10_01_error												:= m01_rs1_r4._10_TT_01_Error,         
			TT_10_03													:= m01_rs1_r4._10_TT_03,               
			TT_10_03_offset												:= m01_rs1_r4.cart10_front_temp_offset,
			TT_10_03_error												:= m01_rs1_r4._10_TT_03_Error,         
			TT_11_01													:= m01_rs1_r4._11_TT_01,               
			TT_11_01_offset												:= m01_rs1_r4.cart11_front_temp_offset,
			TT_11_01_error												:= m01_rs1_r4._11_TT_01_Error,         
			TT_11_03													:= m01_rs1_r4._11_TT_03,               
			TT_11_03_offset												:= m01_rs1_r4.cart11_front_temp_offset,
			TT_11_03_error												:= m01_rs1_r4._11_TT_03_Error,         
			TT_12_01													:= m01_rs1_r4._12_TT_01,               
			TT_12_01_offset												:= m01_rs1_r4.cart12_front_temp_offset,
			TT_12_01_error												:= m01_rs1_r4._12_TT_01_Error,         
			TT_12_03													:= m01_rs1_r4._12_TT_03,               
			TT_12_03_offset												:= m01_rs1_r4.cart12_front_temp_offset,
			TT_12_03_error												:= m01_rs1_r4._12_TT_03_Error,  

			cart01_front_temp											=> m01_rs1_r4.cart01_front_temp,						
			cart01_front_temp_error 									=> m01_rs1_r4.cart01_front_temp_error,
			cart01_back_temp											=> m01_rs1_r4.cart01_back_temp,
			cart01_back_temp_error 										=> m01_rs1_r4.cart01_back_temp_error,
			cart02_front_temp											=> m01_rs1_r4.cart02_front_temp,						
			cart02_front_temp_error 									=> m01_rs1_r4.cart02_front_temp_error,
			cart02_back_temp											=> m01_rs1_r4.cart02_back_temp,
			cart02_back_temp_error 										=> m01_rs1_r4.cart02_back_temp_error,
			cart03_front_temp											=> m01_rs1_r4.cart03_front_temp,						
			cart03_front_temp_error 									=> m01_rs1_r4.cart03_front_temp_error,
			cart03_back_temp											=> m01_rs1_r4.cart03_back_temp,
			cart03_back_temp_error 										=> m01_rs1_r4.cart03_back_temp_error,
			cart04_front_temp											=> m01_rs1_r4.cart04_front_temp,						
			cart04_front_temp_error 									=> m01_rs1_r4.cart04_front_temp_error,
			cart04_back_temp											=> m01_rs1_r4.cart04_back_temp,
			cart04_back_temp_error 										=> m01_rs1_r4.cart04_back_temp_error,
			cart05_front_temp											=> m01_rs1_r4.cart05_front_temp,						
			cart05_front_temp_error 									=> m01_rs1_r4.cart05_front_temp_error,
			cart05_back_temp											=> m01_rs1_r4.cart05_back_temp,
			cart05_back_temp_error 										=> m01_rs1_r4.cart05_back_temp_error,
			cart06_front_temp											=> m01_rs1_r4.cart06_front_temp,						
			cart06_front_temp_error 									=> m01_rs1_r4.cart06_front_temp_error,
			cart06_back_temp											=> m01_rs1_r4.cart06_back_temp,
			cart06_back_temp_error 										=> m01_rs1_r4.cart06_back_temp_error,
			cart07_front_temp											=> m01_rs1_r4.cart07_front_temp,						
			cart07_front_temp_error 									=> m01_rs1_r4.cart07_front_temp_error,
			cart07_back_temp											=> m01_rs1_r4.cart07_back_temp,
			cart07_back_temp_error 										=> m01_rs1_r4.cart07_back_temp_error,
			cart08_front_temp											=> m01_rs1_r4.cart08_front_temp,						
			cart08_front_temp_error 									=> m01_rs1_r4.cart08_front_temp_error,
			cart08_back_temp											=> m01_rs1_r4.cart08_back_temp,
			cart08_back_temp_error 										=> m01_rs1_r4.cart08_back_temp_error,
			cart09_front_temp											=> m01_rs1_r4.cart09_front_temp,						
			cart09_front_temp_error 									=> m01_rs1_r4.cart09_front_temp_error,
			cart09_back_temp											=> m01_rs1_r4.cart09_back_temp,
			cart09_back_temp_error 										=> m01_rs1_r4.cart09_back_temp_error,
			cart10_front_temp											=> m01_rs1_r4.cart10_front_temp,						
			cart10_front_temp_error 									=> m01_rs1_r4.cart10_front_temp_error,
			cart10_back_temp											=> m01_rs1_r4.cart10_back_temp,
			cart10_back_temp_error 										=> m01_rs1_r4.cart10_back_temp_error,
			cart11_front_temp											=> m01_rs1_r4.cart11_front_temp,						
			cart11_front_temp_error 									=> m01_rs1_r4.cart11_front_temp_error,
			cart11_back_temp											=> m01_rs1_r4.cart11_back_temp,
			cart11_back_temp_error 										=> m01_rs1_r4.cart11_back_temp_error,
			cart12_front_temp											=> m01_rs1_r4.cart12_front_temp,						
			cart12_front_temp_error 									=> m01_rs1_r4.cart12_front_temp_error,
			cart12_back_temp											=> m01_rs1_r4.cart12_back_temp,
			cart12_back_temp_error 										=> m01_rs1_r4.cart12_back_temp_error,       
		                                                        
			inlet_co2_pump												:= m01_rs1_r4.inlet_co2_pump,
			AT_01_pump													=> m01_rs1_r4.AT_01_pump,
			inlet_co2_pump_cmd_status									=> m01_rs1_r4.inlet_co2_pump_cmd_status,
			inlet_co2_sol												:= m01_rs1_r4.inlet_co2_sol,
			AT_01_sol													=> m01_rs1_r4.AT_01_sol,
			inlet_co2_sol_cmd_status									=> m01_rs1_r4.inlet_co2_sol_cmd_status,
			outlet_co2_pump												:= m01_rs1_r4.outlet_co2_pump,
			AT_03_pump													=> m01_rs1_r4.AT_03_pump,
			outlet_co2_pump_cmd_status									=> m01_rs1_r4.outlet_co2_pump_cmd_status,
			outlet_co2_sol												:= m01_rs1_r4.outlet_co2_sol,
			AT_03_sol													=> m01_rs1_r4.AT_03_sol,
			outlet_co2_sol_cmd_status									=> m01_rs1_r4.outlet_co2_sol_cmd_status,
			repres_valve												:= m01_rs1_r4.repres_valve,
			XV_02														=> m01_rs1_r4.XV_02,
			repres_valve_open_cmd_status								=> m01_rs1_r4.repres_valve_open_cmd_status,
			repres_valve_open											:= m01_rs1_r4.repres_valve_open,
			repres_valve_closed											:= m01_rs1_r4.repres_valve_closed,
    	                                                        
			fan_vfd_control												=> m01_rs1_r4.fan_vfd_control,  		
			fan_vfd_target_vel	 		                                => m01_rs1_r4.fan_vfd_target_vel, 
			fan_vfd_enabled	 		                                    => m01_rs1_r4.fan_vfd_enabled, 
			fan_vfd_error		                                        => m01_rs1_r4.fan_vfd_error,
			fan_vfd_output												=> m01_rs1_r4.fan_vfd_output,
			fan_vfd_reset												:= m01_rs1_r4.fan_vfd_reset,
			fan_vfd_enable												:= m01_rs1_r4.fan_vfd_enable,
			fan_vfd_ecat_state											:= m01_rs1_r4.fan_vfd_ecat_state,
			fan_vfd_status												:= m01_rs1_r4.fan_vfd_status,
			fan_vfd														:= m01_rs1_r4.fan_vfd,
			fan_vfd_velocity											:= m01_rs1_r4.fan_vfd_velocity,
			fan_vfd_current												:= m01_rs1_r4.fan_vfd_current,
			fan_vfd_current_amps										=> m01_rs1_r4.fan_vfd_output_current,
			                                                    
			inlet_door_clamps_extend									:= m01_rs1_r4.inlet_door_clamps_extend,
			outlet_door_clamps_extend									:= m01_rs1_r4.outlet_door_clamps_extend,
			inlet_door_clamps_retract									:= m01_rs1_r4.inlet_door_clamps_retract,
			outlet_door_clamps_retract									:= m01_rs1_r4.outlet_door_clamps_retract,
			                                                    
			extend_clamps												:= extend_clamps,
			retract_clamps												:= retract_clamps,
			                                                    
			inlet_door_left_clamps_extend								=> m01_rs1_r4.XV_01_Left_Extend_Solenoid_Valve,
			inlet_door_right_clamps_extend								=> m01_rs1_r4.XV_01_Right_Extend_Solenoid_Valve,
			outlet_door_left_clamps_extend								=> m01_rs1_r4.XV_03_Left_Extend_Solenoid_Valve,
			outlet_door_right_clamps_extend								=> m01_rs1_r4.XV_03_Right_Extend_Solenoid_Valve,
			inlet_door_left_clamps_retract								=> m01_rs1_r4.XV_01_Left_Retract_Solenoid_Valve,
			inlet_door_right_clamps_retract								=> m01_rs1_r4.XV_01_Right_Retract_Solenoid_Valve,
			outlet_door_left_clamps_retract								=> m01_rs1_r4.XV_03_Left_Retract_Solenoid_Valve,
			outlet_door_right_clamps_retract							=> m01_rs1_r4.XV_03_Right_Retract_Solenoid_Valve,
    	                                                        
			inlet_door_left_clamps_extended								:= m01_rs1_r4.inlet_door_left_clamps_extended_ls,  
			inlet_door_right_clamps_extended							:= m01_rs1_r4.inlet_door_right_clamps_extended_ls, 
			outlet_door_left_clamps_extended							:= m01_rs1_r4.outlet_door_left_clamps_extended_ls, 
			outlet_door_right_clamps_extended							:= m01_rs1_r4.outlet_door_right_clamps_extended_ls,
			                                                    
			inlet_door_open												:= m01_rs1_r4.inlet_door_open,
			inlet_door_close											:= m01_rs1_r4.inlet_door_close,
			outlet_door_open											:= m01_rs1_r4.outlet_door_open,
			outlet_door_close											:= m01_rs1_r4.outlet_door_close,
			                                                    
			open_doors													:= open_doors,
			close_doors													:= close_doors,
			                                                    
			open_inlet_door												=> m01_rs1_r4.XV_01_Door_Open_Solenoid_Valve,
			close_inlet_door											=> m01_rs1_r4.XV_01_Door_Close_Solenoid_Valve,
			open_outlet_door											=> m01_rs1_r4.XV_03_Door_Open_Solenoid_Valve,
			close_outlet_door											=> m01_rs1_r4.XV_03_Door_Close_Solenoid_Valve,
			                                                    
			inlet_door_left_open										:= m01_rs1_r4.inlet_door_left_open_ls, 
			inlet_door_right_open										:= m01_rs1_r4.inlet_door_right_open_ls, 
			outlet_door_left_open										:= m01_rs1_r4.outlet_door_left_open_ls, 
			outlet_door_right_open										:= m01_rs1_r4.outlet_door_right_open_ls,
			inlet_door_left_closed										:= m01_rs1_r4.inlet_door_left_closed_ls, 
			inlet_door_right_closed										:= m01_rs1_r4.inlet_door_right_closed_ls, 
			outlet_door_left_closed										:= m01_rs1_r4.outlet_door_left_closed_ls, 
			outlet_door_right_closed									:= m01_rs1_r4.outlet_door_right_closed_ls,
			                                                    
			vacuum_cooling_high_temp_count								=> m01_rs1_r4.vacuum_cooling_high_temp_count,
			adsorption_high_temp_count									=> m01_rs1_r4.adsorption_high_temp_count,
			desorption_high_temp_count									=> m01_rs1_r4.desorption_air_high_temp_count);
END_ACTION

END_PROGRAM

// ---- POUs/Reactor_Set_Function_Blocks/FB_Reactor_Set.TcPOU
FUNCTION_BLOCK FB_Reactor_Set
VAR_IN_OUT
	U																	: Utility;
	R_S																	: Reactor_Set;
	Stop_Reactor_Set													: BOOL;
	Clear_Reactor_Set_Pause												: BOOL;
	test_error															: BOOL;
END_VAR
VAR_INPUT
	RS_Name																: STRING;
	Cycle_Mode															: STRING;
	Fan_Setpoint														: REAL;
	RS_number															: INT;
//	Evac_Service_Acked													: BOOL;
	Evac_Service_Assigned												: BOOL;
	Steam_Service_Assigned												: BOOL;
END_VAR
VAR_OUTPUT
	Cycle_Stage															: STRING;
	Remaining_Time														: REAL;
	Current_Step														: INT;
	Machine_State														: INT;
	Status																: INT;
	Process_Running														: BOOL;
	Pause_Reactor_Set													: BOOL;
	Reactor_Set_Stopped													: BOOL;
	Repressurization_Running											: BOOL;
	Adsorption_Running													: BOOL;
	Evacuation_Running													: BOOL;
	Desorption_Running													: BOOL;
	Utility_Error														: BOOL;
	Stop_M01_RS															: BOOL;
	Cancel_Reactor_Set													: BOOL;
	Cancel_All_Reactor_Sets												: BOOL;
	Process_Complete													: BOOL;
	Done																: BOOL;
	Evac_Service_Req														: BOOL;
	Steam_Service_Req													: BOOL;
END_VAR

VAR
	eState																: E_MachineState;
	i																	: INT;
	iStatePointer														: INT;
	iLength																: INT;
	iStateMode															: ARRAY[0..9] OF INT;
	
	sSafeShutdownError1													: STRING;
	sSafeShutdownError2													: STRING;
	sSafeShutdownError3													: STRING;
	sUtilityError														: STRING;
	sReactorError														: STRING;
	sCancelError														: STRING;
	sPauseError															: STRING;
	sRetryError															: STRING;
	sLastRetryError														: STRING;
	sError																: STRING;
	sMessage															: STRING;
	sLeakageAcceptable													: STRING;
	sLeakageUnacceptable												: STRING;

	rTime																: REAL;
	rTime1																: REAL;
	rTime2																: REAL;
	rTime3																: REAL;
	rSP1																: REAL;
	rSP2																: REAL;
	rSP3																: REAL;
	rR1SavedPressure													: REAL;
	rR2SavedPressure													: REAL;
	rR3SavedPressure													: REAL;
	rR4SavedPressure													: REAL;
	rIncrementalMove													: REAL;
	rPosition															: REAL;
	
	tTime																: TIME;
	
	iStep																: INT;
	i4Step																: INT;
	i5Step																: INT;
	i6Step																: INT;
	i7Step																: INT;
	iSS1Step															: INT;
	iSS2Step															: INT;
	iSS3Step															: INT;
	iStartStep															: INT;
	iStatus																: INT;
	iRestartProcess														: INT;
	iErrorProcess														: INT;
	iRestartStep														: INT;
	iRetryCount															: INT;
	iR1Leakage															: INT;
	iR2Leakage															: INT;
	iR3Leakage															: INT;
	iR4Leakage															: INT;
	iCycleCount															: INT;
	iMaxSorbentTempErrorCount											: INT;
	iSSType																: INT;
	iSafeShutdown														: INT;
	iSafeShutdownRS														: INT;

	bMultiProcess														: BOOL;
	bEndProcess															: BOOL;
	bSPAdjust															: BOOL;
	bPaused																: BOOL;
	bClearingCycle														: BOOL;
	bRepressurizationDone												: BOOL;
	bAdsorptionDone														: BOOL;
	bEvacuationDone														: BOOL;
	bDesorptionDone									        			: BOOL;
	bPass1																: BOOL;
	bPass2																: BOOL;
	bPass3																: BOOL;
	bPass4																: BOOL;
	bPass5																: BOOL;
	bPass6																: BOOL;
	bLowPressure														: BOOL;
	bStop																: BOOL;
	bTimer1																: BOOL;
	bTimer2																: BOOL;
	bTimer3																: BOOL;
	bRunning															: BOOL;
	bDrainError															: BOOL;
	bPumpOn																: BOOL;
	bPumpTimeOut														: BOOL;									
	bDrainResetToLSL													: BOOL;
	bProcessStarted														: BOOL;
	bEvacuationRSError													: BOOL;
	bDesorptionRSError													: BOOL;
	bDesorptionErrorCheck												: BOOL;
	bStopAfterDesorption												: BOOL;
	bStopAfterEvacuation												: BOOL;
	bSafeShutdownOn														: BOOL;
	
	rtrigStart															: R_TRIG;
	rtrigPaused															: R_TRIG;
	rtrigHolding														: R_TRIG;
	rtrigIdle															: R_TRIG;
	rtrigRepressurization												: R_TRIG;
	rtrigAdsorption														: R_TRIG;
	rtrigEvacuation														: R_TRIG;
	rtrigDesorption														: R_TRIG;
	rtrigDrainLSHOn														: R_TRIG;
	
	tonTimer1															: TON;
	tonTimer2															: TON;
	tonTimer3															: TON;
	tonPause															: TON;
	tonDrain															: TON;
	tonProcess															: TON;
	
	tRestartTime														: TIME;
END_VAR

// Phase 0 - FB_Reactor_Set
// Rev 1.0 - May 13, 2024

A_Clear_Variables();

iLength																	:= LEN(Cycle_Mode);
rtrigStart(CLK:= iLength > 0);
IF rtrigStart.Q AND iSS1Step = 0 AND iSS2Step = 0 AND iSS3Step = 0 THEN
	IF Cycle_Mode = '0' THEN
		bClearingCycle													:= TRUE;											// This acts as if the cycle ran so the reactor set cycle counter will stay in sync with the other reactor sets		
	ELSE
		bProcessStarted													:= TRUE;
		IF Pause_Reactor_Set THEN
			bPaused														:= TRUE;
		ELSE
			iStartStep													:= 1;
			Process_Running												:= TRUE;
			FOR i := 1 TO iLENGTH DO
				iStateMode[i]											:= STRING_TO_INT(MID(Cycle_Mode, 1, i));
			END_FOR
			bMultiProcess												:= iLength > 1;
			IF bMultiProcess AND iRestartProcess > 0 THEN
				iStatePointer											:= iRestartProcess;
				iStartStep												:= iRestartStep;
				iRestartProcess											:= 0;
				Machine_State											:= eHolding;
			ELSE
				iRestartProcess											:= 0;
				iStatePointer											:= 1;
				Machine_State											:= iStateMode[1];
			END_IF
		END_IF
	END_IF
END_IF

rtrigIdle(				CLK:= eState <= eIdle);
rtrigPaused(			CLk:= bPaused);
rtrigHolding(			CLK:= Machine_State = eHolding);
rtrigRepressurization(	CLK:= Machine_State = eRepressurization);
rtrigAdsorption(		CLK:= Machine_State = eAdsorption);
rtrigEvacuation(		CLK:= Machine_State = eEvacuation);
rtrigDesorption(		CLK:= Machine_State = eDesorption);

IF rtrigPaused.Q THEN
	bPaused																:= FALSE;
	eState																:= ePause;
ELSIF rtrigHolding.Q THEN
	eState																:= eHolding;
ELSIF rtrigRepressurization.Q THEN
	bRepressurizationDone												:= FALSE;
	i4Step																:= iStartStep;
	eState																:= eRepressurization;
ELSIF rtrigAdsorption.Q THEN
	bAdsorptionDone														:= FALSE;
	i5Step																:= iStartStep;
	eState																:= eAdsorption;
ELSIF rtrigEvacuation.Q THEN
	bEvacuationDone														:= FALSE;
	i6Step																:= iStartStep;
	eState																:= eEvacuation;
ELSIF rtrigDesorption.Q THEN
	bDesorptionDone														:= FALSE;
	i7Step																:= iStartStep;
	eState																:= eDesorption;
ELSIF rtrigIdle.Q THEN
	bProcessStarted														:= FALSE;
	eState																:= eIdle;
END_IF


CASE eState OF
	
	eIdle:
		A1_Idle();
		
	eHolding:
		A2_Holding();
		
	eRepressurization:
		IF bRepressurizationDone THEN
			Repressurization_Running									:= FALSE;
			IF bMultiProcess THEN
				eState													:= SEL(bStop, eChangeState, ePause);
			ELSE
				Status													:= SEL(bStop, eRepressurization_Complete, Status);
				eState													:= ePause;
			END_IF
		ELSIF bStop THEN
			Status														:= eStopping_Process;
		ELSE
			Status														:= eRepressurization_Running;
			Repressurization_Running									:= TRUE;
		END_IF

	eAdsorption:
		IF bAdsorptionDone THEN
			Adsorption_Running											:= FALSE;
			IF bMultiProcess THEN
				eState													:= SEL(bStop, eChangeState, ePause);
			ELSE
				Status													:= SEL(bStop, eAdsorption_Complete, Status);
				eState													:= ePause;
			END_IF
		ELSIF bStop THEN
			Status														:= eStopping_Process;
		ELSE
			Status														:= eAdsorption_Running;
			Adsorption_Running											:= TRUE;
		END_IF

	eEvacuation:
		IF bEvacuationDone THEN
			Evacuation_Running											:= FALSE;
			IF bMultiProcess THEN
				eState													:= SEL(bStop, eChangeState, ePause);
			ELSE
				Status													:= SEL(bStop, eEvacuation_Complete, Status);
				eState													:= ePause;
			END_IF
		ELSIF bStop THEN
			Status														:= eStopping_Process;
		ELSE
			Status														:= eEvacuation_Running;
			Evacuation_Running											:= TRUE;
		END_IF
		
	eDesorption:
		IF bDesorptionDone THEN
			Desorption_Running											:= FALSE;
			IF bMultiProcess THEN
				eState													:= SEL(bStop, eChangeState, ePause);
			ELSE
				Status													:= SEL(bStop, eDesorption_Complete, Status);
				eState													:= ePause;
			END_IF
		ELSIF bStop THEN
			Status														:= eStopping_Process;
		ELSE
			Status														:= eDesorption_Running;
			Desorption_Running											:= TRUE;
		END_IF
		
	eChangeState:
		iStatePointer													:= iStatePointer + 1;
		IF iStatePointer > iLength THEN
			Process_Complete											:= TRUE;
			Done														:= TRUE;
			eState														:= eIdle;
		ELSIF iStateMode[iStatePointer] = 0 THEN
			Status														:= eStopping_Process;
			bStop														:= TRUE;
			bMultiProcess												:= FALSE;
			eState														:= ePause;
		ELSE
			Machine_State												:= iStateMode[iStatePointer];
		END_IF
	
	ePause:
		Machine_State													:= ePause;
		IF tonPause.Q THEN
			IF iSSType = 1 THEN
				iSSType													:= 0;
				iSS1Step												:= 1;
				eState													:= eSafeShutdown1;
			ELSIF iSSType = 2 THEN
				iSSType													:= 0;
				iSS2Step												:= 1;
				eState													:= eSafeShutdown2;
			ELSIF iSSType = 3 THEN
				iSSType													:= 0;
				iSS3Step												:= 1;
				eState													:= eSafeShutdown3;
			ELSE
				Done													:= TRUE;
				eState													:= eIdle;
			END_IF
		END_IF
		
	eSafeShutdown1:
		Machine_State													:= eSafeShutdown1;
		A_SafeShutdown1_Test();
		IF iSS1Step	= 0 THEN
			eState														:= ePause;
		END_IF
	
	eSafeShutdown2:
		Machine_State													:= eSafeShutdown2;
		A_SafeShutdown2_Test();
		IF iSS2Step	= 0 THEN
			eState														:= ePause;
		END_IF
	
	eSafeShutdown3:
		Machine_State													:= eSafeShutdown3;
		A_SafeShutdown3_Test();
		IF iSS3Step	= 0 THEN
			eState														:= ePause;
		END_IF
	
END_CASE

bRunning																:= eState >= eHolding AND eState <= ePause;

//A4_Repressurization_Test();
A4_Repressurization_Test_Auto();
//A5_Adsorption_Test();
A5_Adsorption_Test_Auto();
//A6_Evacuation_Test();
A6_Evacuation_Test_Auto();
//A7_Desorption_Test();
A7_Desorption_Test_Auto();
//A_Drain_Reactor_Set();

tonTimer1(IN:= bTimer1, PT:= REAL_TO_TIME(rTime1));
tonTimer2(IN:= bTimer2, PT:= REAL_TO_TIME(rTime2));
tonTimer3(IN:= bTimer3, PT:= REAL_TO_TIME(rTime3));

Remaining_Time															:= 0;
IF Process_Running THEN
	IF bTimer1 THEN
		Remaining_Time													:= rTime1 - TIME_TO_REAL(tonTimer1.ET);
	ELSIF bTimer2 THEN
		Remaining_Time													:= rTime2 - TIME_TO_REAL(tonTimer2.ET);
	ELSIF bTimer3 THEN
		Remaining_Time													:= rTime3 - TIME_TO_REAL(tonTimer3.ET);
	END_IF
END_IF

tonPause(IN:= eState = ePause, PT:= _TIMEOUT_RESET);
tonProcess(IN:= bProcessStarted, PT:= T#10H);

ACTION A_Check_Process:
// Phase 0 - FB_Reactor_Set.A_ClearProcess
// Rev 1.0 - May 13, 2024

Current_Step															:= iStep;
bEndProcess																:= FALSE;
IF Stop_Reactor_Set THEN																									// Reactor Set can be stopped both internally and externally
	Stop_Reactor_Set													:= FALSE;											// Clear flag
	bEndProcess															:= TRUE;											// Set flag to end process
ELSE
	IF sSafeShutdownError1 <> '' THEN
		iSSType															:= 1; 	
		sError															:= sSafeShutdownError1;
		sSafeShutdownError1												:= '';
		sMessage														:= gsSafeShutdown1;
		bEndProcess														:= TRUE;
	ELSIF sSafeShutdownError2 <> '' THEN
		iSSType															:= 2; 	
		sError															:= sSafeShutdownError2;
		sSafeShutdownError2												:= '';
		sMessage														:= gsSafeShutdown2;
		bEndProcess														:= TRUE;
	ELSIF sSafeShutdownError3 <> '' THEN
		iSSType															:= 3; 	
		sError															:= sSafeShutdownError3;
		sSafeShutdownError3												:= '';
		sMessage														:= gsSafeShutdown3;
		bEndProcess														:= TRUE;
	ELSIF sUtilityError <> '' THEN																							//@ Times used - 3
		sError															:= sUtilityError;
		Utility_Error													:= TRUE;
		iStep															:= 98;
	ELSIF sReactorError <> '' THEN																							//@ Times used - 43
		sError															:= sReactorError;
  		bEndProcess														:= TRUE;
	ELSIF sPauseError <> '' THEN																							//@ Times used - 2
		sError															:= sPauseError;
		iRestartProcess													:= F_SetProcess(eRepressurization, Cycle_Mode);		// Set restart to Repressurization
		Pause_Reactor_Set												:= TRUE;
		bEndProcess														:= TRUE;
	ELSIF sRetryError <> '' THEN																							//@ Times used - 1
		sError															:= sRetryError;
		tRestartTime													:= tonProcess.ET;									// Save time to start retry attempt
		iRestartProcess													:= iStatePointer;									// Get current process machine state
		iErrorProcess													:= iStatePointer;									// Save machine state for later reference
		IF sError = sLastRetryError THEN																					// If the same error occured,
			iRetryCount													:= iRetryCount + 1;									// increment the retry counter
			IF iRetryCount >= _RETRY_ATTEMPTS THEN																			// If retry attempts have maxed out,
				sMessage												:= gsUserProcessRestart;							// let user know in the message	they must now manually restart	
				iRestartProcess											:= 0;												// Clear the restart variables
				iRetryCount												:= 0;
				sLastRetryError											:= '';
				Pause_Reactor_Set										:= TRUE;
				Stop_M01_RS												:= TRUE;
			END_IF
		ELSE
			iRetryCount													:= 1;												// Increment retry counter
			sLastRetryError												:= sError;											// Save error message for later reference	
		END_IF
		bEndProcess														:= TRUE;
	END_IF
	IF iErrorProcess > 0 AND iErrorProcess <> iStatePointer THEN
		iRestartProcess													:= 0;
		iErrorProcess													:= 0;
		iRetryCount														:= 0;
		iRestartStep													:= 1;
		sLastRetryError													:= '';
	END_IF
	IF sError <> '' THEN
		P_Alarms.M_Add_Alarm(RS_Name, F_Concat3(Cycle_Stage, ' ', sError), sMessage);
		sError															:= '';
	END_IF
END_IF

IF bEndProcess THEN
	bTimer1								 								:= FALSE;
	bTimer2								 								:= FALSE;
	bStop																:= TRUE;
	Stop_M01_RS															:= TRUE;											// Stop Reactor in P_M01.A_AutoMode
	iStep																:= SEL(bMultiProcess, 80, 90);
	Evac_Service_Req													:= FALSE;
	Steam_Service_Req													:= FALSE;
END_IF
END_ACTION

ACTION A_Clear_Variables:
// Phase 0 - FB_Reactor_Set.A_Clear_Variables
// Rev 1.0 - June 3, 2024

R_S.extend_all_clamps													:= FALSE;
R_S.retract_all_clamps													:= FALSE;
R_S.open_all_doors														:= FALSE;
R_S.close_all_doors														:= FALSE;
R_S.close_all_valves													:= FALSE;
R_S.co2_sensors_off														:= FALSE;
R_S.co2_inside_sensors_on												:= FALSE;
R_S.co2_outside_sensors_on												:= FALSE;
R_S.open_repres_valves													:= FALSE;
R_S.close_repres_valves													:= FALSE;
Utility_Error															:= FALSE;
//Stop_Reactor_Set														:= FALSE;
Cancel_Reactor_Set														:= FALSE;
Cancel_All_Reactor_Sets													:= FALSE;
Stop_M01_RS																:= FALSE;
sSafeShutdownError1														:= '';
sSafeShutdownError2														:= '';
sSafeShutdownError3														:= '';
sUtilityError															:= '';
sReactorError															:= '';
sPauseError																:= '';
sRetryError																:= '';
IF Clear_Reactor_Set_Pause THEN
	Clear_Reactor_Set_Pause												:= FALSE;
	Pause_Reactor_Set													:= FALSE;
END_IF
IF NOT U.auto_mode_on THEN
	iMaxSorbentTempErrorCount											:= 0;
	iCycleCount															:= 0;	
END_IF
END_ACTION

ACTION A_Drain_Reactor_Set:
// Phase 0 - FB_Reactor_Set.A_Drain_Reactor_Set
// Rev 1.0 - March 8, 2024

IF gbDrainageOn THEN																										// 4.1.1
	
	bLowPressure														:= NOT R_S.R1_reactor_pres_error AND R_S.R1_reactor_pres < u01.SP_drainage_function_cutoff_pressure;
	bLowPressure														:= bLowPressure AND NOT R_S.R2_reactor_pres_error AND R_S.R2_reactor_pres < u01.SP_drainage_function_cutoff_pressure;
	bLowPressure														:= bLowPressure AND NOT R_S.R3_reactor_pres_error AND R_S.R3_reactor_pres < u01.SP_drainage_function_cutoff_pressure;
	bLowPressure														:= bLowPressure AND NOT R_S.R4_reactor_pres_error AND R_S.R4_reactor_pres < u01.SP_drainage_function_cutoff_pressure;
	IF bLowPressure THEN
		bPumpOn															:= FALSE;											// 1.b
	ELSE
		rtrigDrainLSHOn(CLK:= R_S.condensate_lsh);
		IF rtrigDrainLSHOn.Q THEN
			bDrainResetToLSL											:= TRUE;
		END_IF
		IF bDrainResetToLSL AND R_S.condensate_lsl THEN
			bPumpOn														:= TRUE;
		ELSE
			bPumpOn														:= FALSE;
			bDrainResetToLSL											:= FALSE;
		END_IF
	END_IF
	
	IF tonDrain.Q THEN
		P_Alarms.M_Add_Alarm(RS_Name, gsReactorDrainError, gsProcessStopsAtEOC);
		bPumpOn															:= FALSE;
		bDrainError														:= TRUE;
		Cancel_Reactor_Set												:= TRUE; 
	END_IF
	tonDrain(IN:= R_S.condensate_lsh AND NOT bDrainError, PT:= REAL_TO_TIME(u01.SP_maximum_duration_to_drain_reactor_set * _SECONDS));
	bPumpTimeOut														:= tonDrain.ET > REAL_TO_TIME(u01.SP_duration_to_drain_reactor_set * _SECONDS);
	
	IF NOT R_S.condensate_lsh THEN
		bDrainError														:= FALSE;
	END_IF

	R_S.condensate_pump													:= bPumpOn AND NOT bDrainError AND NOT bPumpTimeOut;
	
END_IF
END_ACTION

ACTION A_SafeShutdown1:
// Phase 0 - FB_Reactor_Set.A_SafeShutdown1
// Rev 1.0 - May 10, 2024

CASE iSS1Step OF
	
	0:	;
		
	1:	
		sError															:= '';
		sMessage														:= gsUnableToEvacuateReactorSet;
		rTime2															:= m01.SP_evacuation_duration * 3 * _MINUTES;
		iSS1Step														:= iSS1Step + 1;
		
	2:
		bTimer2															:= TRUE;											// 1
		Cycle_Stage														:= 'evacuation.safe_shutdown_1';					// 1.a
		U.dead_air_vacuum_pump											:= TRUE;											// 2
		R_S.close_all_doors												:= TRUE;											// 3
		rTime1															:= m01.SP_doorsopenclose_timedelay * _MINUTES;
		iSS1Step														:= iSS1Step + 1;
		
	3:
		bTimer1															:= TRUE;
		IF R_S.all_doors_closed THEN
			bTimer1														:= FALSE;
			R_S.close_repres_valves										:= TRUE;											// 4
			rTime1														:= _VALVE_TIME;
			iSS1Step													:= iSS1Step + 1;
		ELSIF tonTimer1.Q THEN
			bTimer1														:= FALSE;
			sError														:= gsDoorsNotClosedError;
			iSS1Step													:= 80;
		END_IF
		
	4:
		bTimer1															:= TRUE;
		IF R_S.repres_valve_error = '' THEN
			bTimer1														:= FALSE;
			IF R_S.all_clamps_extended THEN
				iSS1Step												:= iSS1Step + 2;
			ELSE
				R_S.extend_all_clamps									:= TRUE;											// 5
				rTime1													:= m01.SP_extend_wallace_clamp_duration * _MINUTES;
				iSS1Step												:= iSS1Step + 1;
			END_IF
		ELSIF tonTimer1.Q THEN
			bTimer1														:= FALSE;
			sError														:= gsRepressurizationValveError;
			iSS1Step													:= 80;
		END_IF
		
	5:
		bTimer1															:= TRUE;
		IF tonTimer1.Q THEN
			bTimer1														:= FALSE;
			iSS1Step													:= iSS1Step + 1;
		END_IF
		
	6:
		IF U.dead_air_line_pres < R_S.average_reactor_pressure THEN															// 6
			R_S.dead_air_valve											:= TRUE;											// 7
			iSS1Step													:= iSS1Step + 1;
		ELSIF TIME_TO_REAL(tonTimer2.ET) > (m01.SP_evacuation_duration * 2 * _MINUTES) THEN
			sError														:= 	gsUnableToEvacuateLinesError;
			iSS1Step													:= 80;
		END_IF
		
	7:
		IF tonTimer2.Q THEN																									// 8
			bTimer2														:= FALSE;
			IF R_S.average_reactor_pressure >= m01.SP_evacuation_unacceptable_pressure THEN									// 8.c
				sError													:= gsInsufficientVacuumPressureError;
			ELSIF R_S.average_reactor_pressure > m01.SP_evacuation_ideal_pressure THEN										// 8.b
				sError													:= gsVacuumPressureAcceptableBotNotIdealError;
			END_IF
			iSS1Step													:= 80;												// else 8.a
		END_IF
		
	80:
		R_S.dead_air_valve												:= FALSE;											// 9
		U.dead_air_vacuum_pump											:= FALSE;											// 10
		bTimer2															:= FALSE;											// 11
		R_S.co2_sensors_off												:= TRUE;											// 12
		IF sError <> '' THEN
			P_Alarms.M_Add_Alarm(RS_Name, sError, sMessage);
		END_IF
		//Stop_Reactor_Set												:= TRUE;
		iSS1Step														:= 0;												// 13
		
END_CASE
END_ACTION

ACTION A_SafeShutdown1_Test:
// Phase 0 - FB_Reactor_Set.A_SafeShutdown1_Test
// Rev 1.0 - May 10, 2024

CASE iSS1Step OF
	
	0:	;
		
	1:	
		Cycle_Stage														:= 'ss_1';
		rTime1															:= 5 * _SECONDS;
		iSS1Step														:= iSS1Step + 1;
		
	2:
		bTimer1															:= TRUE;
		IF tonTimer1.Q THEN
			bTimer1														:= FALSE;
			iSS1Step													:= 80;
		END_IF
		
	80:
		//Stop_Reactor_Set												:= TRUE;
		iSS1Step														:= 0;
		
END_CASE
END_ACTION

ACTION A_SafeShutdown2:
// Phase 0 - FB_Reactor_Set.A_SafeShutdown2
// Rev 1.0 - May 10, 2024

CASE iSS2Step OF
	
	0:	;
		
	1:	
		sError															:= '';
		sMessage														:= gsUnableToEvacuateReactorSet;
		rTime2															:= m01.SP_evacuation_duration * 3 * _MINUTES;
		iSS2Step														:= iSS2Step + 1;
		
	2:
		bTimer2															:= TRUE;											// 1
		Cycle_Stage														:= 'evacuation.safe_shutdown_2';					// 1.a
		R_S.close_all_doors												:= TRUE;											// 2
		rTime1															:= m01.SP_doorsopenclose_timedelay * _MINUTES;
		iSS2Step														:= iSS2Step + 1;
		
	3:
		bTimer1															:= TRUE;
		IF R_S.all_doors_closed THEN
			bTimer1														:= FALSE;
			R_S.close_repres_valves										:= TRUE;											// 3
			rTime1														:= _VALVE_TIME;
			iSS2Step													:= iSS2Step + 1;
		ELSIF tonTimer1.Q THEN
			bTimer1														:= FALSE;
			sError														:= gsDoorsNotClosedError;
			iSS2Step													:= 80;
		END_IF
		
	4:
		bTimer1															:= TRUE;
		IF R_S.repres_valve_error = '' THEN
			bTimer1														:= FALSE;
			IF R_S.all_clamps_extended THEN
				iSS2Step												:= iSS2Step + 2;
			ELSE
				R_S.extend_all_clamps									:= TRUE;											// 4
				rTime1													:= m01.SP_extend_wallace_clamp_duration * _MINUTES;
				iSS2Step												:= iSS2Step + 1;
			END_IF
		ELSIF tonTimer1.Q THEN
			bTimer1														:= FALSE;
			sError														:= gsRepressurizationValveError;
			iSS2Step													:= 80;
		END_IF
		
	5:
		bTimer1															:= TRUE;
		IF tonTimer1.Q THEN
			bTimer1														:= FALSE;
			iSS2Step													:= iSS2Step + 1;
		END_IF
		
	6:
		U.product_condenser												:= TRUE;											// 5
		U.product_vacuum_outlet_isolation_valve							:= TRUE;											// 6
		U.product_vacuum_bypass_valve									:= TRUE;											// 7
		U.product_vacuum_pump_isolation_valve							:= TRUE;											// 8
		U.product_vacuum_backfeed_valve									:= _CLOSED;											// 9
		U.product_vacuum_pump_vfd										:= u01.SP_product_vacuum_running_vfd_percent;		// 10
		U.cooling_line_pre_condenser_valve								:= TRUE;											// 11
		iSS2Step														:= iSS2Step + 1;

	7:	
		IF U.post_condenser_line_pres < R_S.average_reactor_pressure THEN													// 12
			R_S.cooling_valve											:= TRUE;											// 13
			iSS2Step													:= iSS2Step + 1;
		ELSIF TIME_TO_REAL(tonTimer2.ET) > (m01.SP_evacuation_duration * 2 * _MINUTES) THEN					
			sError														:= 	gsUnableToEvacuateLinesError;
			iSS2Step													:= 80;
		END_IF
		
	8:
		IF tonTimer2.Q THEN																									// 14
			bTimer2														:= FALSE;
			IF R_S.average_reactor_pressure >= m01.SP_evacuation_unacceptable_pressure THEN									// 14.c
				sError													:= gsInsufficientVacuumPressureError;
				sMessage												:= gsSorbentDamaged;
			ELSIF R_S.average_reactor_pressure > m01.SP_evacuation_ideal_pressure THEN										// 14.b
				sError													:= gsVacuumPressureAcceptableBotNotIdealError;
			END_IF
			iSS2Step													:= 80;												// else 14.a
		END_IF
		
	80:
		R_S.cooling_valve												:= FALSE;											// 15
		U.product_vacuum_pump_vfd										:= u01.SP_product_vacuum_idle_vfd_percent;			// 16
		U.product_vacuum_outlet_isolation_valve							:= FALSE;											// 17
		U.product_vacuum_bypass_valve									:= FALSE;
		U.product_vacuum_pump_isolation_valve							:= FALSE;
		U.cooling_line_pre_condenser_valve								:= FALSE;
		U.product_condenser												:= FALSE;											// 18
		U.dead_air_vacuum_pump											:= FALSE;
		bTimer2															:= FALSE;											// 19
		R_S.co2_sensors_off												:= TRUE;											// 20
		IF sError <> '' THEN
			P_Alarms.M_Add_Alarm(RS_Name, sError, sMessage);
		END_IF
		//Stop_Reactor_Set												:= TRUE;
		iSS2Step														:= 0;												// 21
		
END_CASE
END_ACTION

ACTION A_SafeShutdown2_Test:
// Phase 0 - FB_Reactor_Set.A_SafeShutdown2_Test
// Rev 1.0 - May 13, 2024

CASE iSS2Step OF
	
	0:	;
		
	1:	
		Cycle_Stage														:= 'ss_2';
		rTime1															:= 5 * _SECONDS;
		iSS2Step														:= iSS2Step + 1;
		
	2:
		bTimer1															:= TRUE;
		IF tonTimer1.Q THEN
			bTimer1														:= FALSE;
			iSS2Step													:= 80;
		END_IF
		
	80:
		//Stop_Reactor_Set												:= TRUE;
		iSS2Step														:= 0;
		
END_CASE
END_ACTION

ACTION A_SafeShutdown3:
// Phase 0 - FB_Reactor_Set.A_SafeShutdown3
// Rev 1.0 - May 10, 2024

CASE iSS3Step OF
	
	0:	;
		
	1:	
		sError															:= '';
		sMessage														:= gsUnableToEvacuateReactorSet;
		rTime2															:= m01.SP_evacuation_duration * 3 * _MINUTES;
		iSS3Step														:= iSS3Step + 1;
		
	2:
		bTimer2															:= TRUE;											// 1
		Cycle_Stage														:= 'evacuation.safe_shutdown_3';					// 1.a
		R_S.close_all_doors												:= TRUE;											// 2
		rTime1															:= m01.SP_doorsopenclose_timedelay * _MINUTES;
		iSS3Step														:= iSS3Step + 1;
		
	3:
		bTimer1															:= TRUE;
		IF R_S.all_doors_closed THEN
			bTimer1														:= FALSE;
			R_S.close_repres_valves										:= TRUE;											// 3
			rTime1														:= _VALVE_TIME;
			iSS3Step													:= iSS3Step + 1;
		ELSIF tonTimer1.Q THEN
			bTimer1														:= FALSE;
			sError														:= gsDoorsNotClosedError;
			iSS3Step													:= 80;
		END_IF
		
	4:
		bTimer1															:= TRUE;
		IF R_S.repres_valve_error = '' THEN
			bTimer1														:= FALSE;
			R_S.extend_all_clamps										:= TRUE;											// 4
			rTime1														:= m01.SP_extend_wallace_clamp_duration * _MINUTES;
			iSS3Step													:= iSS3Step + 1;
		ELSIF tonTimer1.Q THEN
			bTimer1														:= FALSE;
			sError														:= gsRepressurizationValveError;
			iSS3Step													:= 80;
		END_IF

	5:
		bTimer1															:= TRUE;
		IF tonTimer1.Q THEN
			bTimer1														:= FALSE;
			U.dead_air_vacuum_pump										:= TRUE;											// 5
			iSS3Step													:= iSS3Step + 1;
		END_IF
	
	6:
		IF U.dead_air_line_pres < R_S.average_reactor_pressure THEN															// 6
			R_S.dead_air_valve											:= TRUE;											// 7
			iSS3Step													:= iSS3Step + 1;
		ELSIF TIME_TO_REAL(tonTimer2.ET) > (m01.SP_evacuation_duration * 2 * _MINUTES) THEN
			sError														:= 	gsUnableToEvacuateLinesError;
			iSS3Step													:= 80;
		END_IF
		
	7:
		IF tonTimer2.Q THEN																									// 8
			bTimer2														:= FALSE;
			IF R_S.average_reactor_pressure >= m01.SP_evacuation_unacceptable_pressure THEN									// 8.c
				sError													:= gsInsufficientVacuumPressureError;
				sMessage												:= gsSorbentDamaged;
			ELSIF R_S.average_reactor_pressure > m01.SP_evacuation_ideal_pressure THEN										// 8.b
				sError													:= gsVacuumPressureAcceptableBotNotIdealError;
			END_IF
			iSS3Step													:= 80;												// else 8.a
		END_IF
		
	80:
		R_S.dead_air_valve												:= FALSE;											// 9
		U.dead_air_vacuum_pump											:= FALSE;											// 10
		bTimer2															:= FALSE;											// 11
		R_S.co2_sensors_off												:= TRUE;											// 12
		IF sError <> '' THEN
			P_Alarms.M_Add_Alarm(RS_Name, sError, sMessage);
		END_IF
		//Stop_Reactor_Set												:= TRUE;
		iSS3Step														:= 0;												// 13
		
END_CASE
END_ACTION

ACTION A_SafeShutdown3_Test:
// Phase 0 - FB_Reactor_Set.A_SafeShutdown3_Test
// Rev 1.0 - May 13, 2024

CASE iSS3Step OF
	
	0:	;
		
	1:	
		Cycle_Stage														:= 'ss_3';
		rTime1															:= 5 * _SECONDS;
		iSS3Step														:= iSS3Step + 1;
		
	2:
		bTimer1															:= TRUE;
		IF tonTimer1.Q THEN
			bTimer1														:= FALSE;
			iSS3Step													:= 80;
		END_IF
		
	80:
		//Stop_Reactor_Set												:= TRUE;
		iSS3Step														:= 0;
		
END_CASE
END_ACTION

ACTION A1_Idle:
// Phase 0 - FB_Reactor_Set.A1_Idle
// Rev 1.0 - May 8, 2024

Machine_State															:= eIdle;
Cycle_Stage																:= 'idle.idle';
sError																	:= '';
i4Step																	:= 0;
i5Step																	:= 0;
i6Step																	:= 0;
i7Step																	:= 0;
iSS1Step																:= 0;
Current_Step															:= 0;
Remaining_Time															:= 0;
Current_Step															:= 0;
Status																	:= 0;
bMultiProcess															:= FALSE;
bTimer1																	:= FALSE;
bTimer2																	:= FALSE;
bStop																	:= FALSE;
bStopAfterDesorption													:= FALSE;
bStopAfterEvacuation													:= FALSE;
Process_Running															:= FALSE;
Process_Complete														:= FALSE;
IF bClearingCycle THEN
	Done																:= TRUE;
	bClearingCycle														:= FALSE;
ELSE
	Done																:= FALSE;
END_IF
END_ACTION

ACTION A2_Holding:
// Phase 0 - FB_Reactor_Set.A2_Holding
// Rev 1.0 - February 29, 2024

IF tonProcess.ET >= tRestartTime THEN
	Machine_State														:= iStateMode[iStatePointer];
END_IF
END_ACTION

ACTION A4_Repressurization:
// Phase 0 - FB_Reactor_Set.A4_Repressurization
// Rev 1.0 - May 13, 2024

CASE i4Step OF
	
	0:	;
		
	1:
		Cycle_Stage														:= 'repressurization.initialize';					// 2.a.i and 4.i
		iRestartStep													:= 1;												// Save pause information if needed
		tRestartTime													:= tonProcess.ET;
		rTime2															:= m01.SP_repressurization_duration * _MINUTES;
		IF R_S.reactor_pressure_error <> '' THEN
			sReactorError												:= R_S.reactor_pressure_error;
			sMessage													:= gsProcessCannotRun;
		ELSIF R_S.inlet_air_high_temp_count > _INLET_AIR_MAX_COUNT THEN
			sReactorError												:= F_Concat3(INT_TO_STRING(R_S.inlet_air_high_temp_count), ' ', gsSorbentTemperatureError);
			sMessage													:= gsProcessCannotRun;
		ELSE
			i4Step														:= i4Step + 1;
		END_IF
			
	2:
		IF NOT bMultiProcess THEN
			IF R_S.average_reactor_pressure_within_ambient THEN																// 2.a.ii
				sReactorError											:= gsReactorsAtAmbientPressure;
				sMessage												:= gsProcessComplete;
			ELSIF NOT R_S.all_clamps_retracted THEN																			// 2.a.iv
				sReactorError											:= gsDoorClampsExtendedError;
				sMessage												:= gsProcessCannotRun;
			ELSE
				i4Step													:= i4Step + 1;
			END_IF
		ELSE
			i4Step														:= i4Step + 1;
		END_IF

	3:
		bTimer2															:= TRUE;											// 4
		U.drainage_on													:= TRUE;											// 5.a
		R_S.close_all_valves											:= TRUE;											// 5.b
		rTime1															:= _VALVE_TIME;
		i4Step															:= i4Step + 1;
		
	4:
		bTimer1															:= TRUE;
		IF R_S.valves_clear THEN
			bTimer1														:= FALSE;
			i4Step														:= i4Step + 1;
		ELSIF tonTimer1.Q THEN
			bTimer1														:= FALSE;
			sReactorError												:= SEL(R_S.Steam_Control_Valve_Closed, gsSteamControlValveError, '');
			sReactorError												:= SEL(R_S.dead_air_valve_clear, gsDeadAirValveError, sReactorError);
			sReactorError												:= SEL(R_S.purge_valve_clear, gsPurgeValveError, sReactorError); 
			sReactorError												:= SEL(R_S.cooling_valve_clear, gsCoolingValveError, sReactorError);
			sReactorError												:= SEL(R_S.steam_header_valve_clear, gsSteamHeaderValveError, sReactorError);
			sMessage													:= gsReactorSetCannotRun;
		END_IF

	5:
		IF R_S.vacuum_cooling_high_temp_count <= _VAC_COOLING_MAX_COUNT THEN												// 5.d
			R_S.co2_outside_sensors_on									:= TRUE;											// 6
			R_S.open_repres_valves										:= TRUE;											// 7
			Cycle_Stage													:= 'repressurization.repressurization';				// 7.i
			rTime1														:= _VALVE_TIME;
			i4Step														:= i4Step + 1;
		ELSE																												// 5.d.i
			sRetryError													:= F_Concat3(INT_TO_STRING(R_S.vacuum_cooling_high_temp_count), ' ', gsSorbentTemperatureError);
			sMessage													:= gsProcessRestart;
		END_IF
		
	6:
		bTimer1															:= TRUE;
		IF R_S.repres_valve_error = '' THEN
			i4Step														:= i4Step + 1;
		ELSIF tonTimer1.Q THEN
			sReactorError												:= R_S.repres_valve_error;
			sMessage													:= gsProcessCannotRun;
		END_IF

	7:
		IF tonTimer2.Q THEN																									// 8
			bTimer2														:= FALSE;
			IF R_S.average_reactor_pressure_within_ambient THEN																// 9
				R_S.co2_sensors_off										:= TRUE;											// 10
				i4Step													:= 99;
			ELSE
				IF R_S.average_reactor_pressure < (m01.SP_vacuum_cooling_target_pressure * _PRESSURE_PERCENT) THEN			// 9.a
					sPauseError											:= gsReactorSetFailedToPressurizeError;
					sMessage											:= gsReactorIsUnderVacuum;
					R_S.close_repres_valves								:= TRUE;
				ELSE																										// 9.b		///! - Narrative not implemented here 
					sReactorError										:= gsReactorSetFailedToPressurizeError;
					sMessage											:= gsProcessCannotContinue;
				END_IF
			END_IF
		END_IF
	
	80:																														// Manual process closing
		Cycle_Stage														:= 'repressurization.stopping';
		R_S.co2_sensors_off												:= TRUE;
		R_S.close_repres_valves											:= TRUE;
		U.drainage_on													:= FALSE;
		rTime1															:= _STOPPING_TIME;
		i4Step															:= i4Step + 1;
		
	81:
		bTimer1															:= TRUE;
		IF tonTimer1.Q THEN
			bTimer1														:= FALSE;
			i4Step														:= 99;
		END_IF
		
	90:																														// Automatic process stopping
		Cycle_Stage														:= 'repressurization.stopping';
		R_S.co2_sensors_off												:= TRUE;
		R_S.close_repres_valves											:= TRUE;
		U.drainage_on													:= FALSE;
		rTime1															:= _STOPPING_TIME;
		i4Step															:= i4Step + 1;
		
	91:
		bTimer1															:= TRUE;
		IF tonTimer1.Q THEN
			bTimer1														:= FALSE;
			i4Step														:= 99;
		END_IF
		
	98:																														// Utility error hold - cleared by P_M01
		i4Step															:= 98;
		
	99:
		bRepressurizationDone											:= TRUE;
		Current_Step													:= 0;
		i4Step															:= 0;
	
END_CASE

IF i4Step > 0 AND i4Step < 80 THEN
	IF bMultiProcess THEN
		IF U.safe_shutdown_error_1 <> '' AND giSafeShutdown1RS = 0 THEN
			sSafeShutdownError1											:= U.safe_shutdown_error_1;
			giSafeShutdown1RS											:= RS_Number;
		ELSIF U.safe_shutdown_error_2 <> '' AND giSafeShutdown23RS = 0 THEN
			sSafeShutdownError2											:= U.safe_shutdown_error_2;
			giSafeShutdown23RS											:= RS_Number;
		ELSIF (giEvacuationErrorRS + giDesorptionErrorRS + giSafeShutdown1RS + giSafeShutdown23RS) > 0 THEN
			Cancel_Reactor_Set											:= TRUE;
		ELSIF U.os_air_unsafe_temp THEN
			Stop_Reactor_Set											:= TRUE;
		END_IF
	END_IF
	iStep																:= i4Step;
	Current_Step														:= iStep;
	A_Check_Process();
	i4Step																:= iStep;
END_IF
END_ACTION

ACTION A4_Repressurization_Test:
// Phase 0 - FB_Reactor_Set.A4_Repressurization_Test
// Rev 1.0 - June 3, 2024

CASE i4Step OF
	
	0:	;
		
	1:
		Cycle_Stage														:= 'repressurization.initialize';					// 2.a.i and 4.i
		iRestartStep													:= 1;												// Save pause information if needed
		tRestartTime													:= tonProcess.ET;
		rTime2															:= m01.SP_repressurization_duration * _MINUTES;
		IF R_S.reactor_pressure_error <> '' THEN
			sReactorError												:= R_S.reactor_pressure_error;
			sMessage													:= gsProcessCannotRun;
		ELSE
			U.drainage_on												:= TRUE;											// 5.a
			R_S.close_all_valves										:= TRUE;											// 5.b
			rTime1														:= _VALVE_TIME;
			i4Step														:= i4Step + 1;
		END_IF
			
	2:
		bTimer1															:= TRUE;
		IF R_S.valves_clear THEN
			bTimer1														:= FALSE;
			i4Step														:= i4Step + 1;
		ELSIF tonTimer1.Q THEN
			bTimer1														:= FALSE;
			sReactorError												:= SEL(R_S.Steam_Control_Valve_Closed, gsSteamControlValveError, '');
			sReactorError												:= SEL(R_S.dead_air_valve_clear, gsDeadAirValveError, sReactorError);
			sReactorError												:= SEL(R_S.purge_valve_clear, gsPurgeValveError, sReactorError); 
			sReactorError												:= SEL(R_S.cooling_valve_clear, gsCoolingValveError, sReactorError);
			sReactorError												:= SEL(R_S.steam_header_valve_clear, gsSteamHeaderValveError, sReactorError);
			sMessage													:= gsReactorSetCannotRun;
		END_IF

	3:
		bTimer2															:= TRUE;
		IF R_S.average_reactor_pressure <= m01.SP_repres_preslimit_clampsretract THEN
			R_S.retract_all_clamps										:= TRUE;
			rTime1														:= 30 * _SECONDS;
			i4Step														:= i4Step + 1;
		ELSIF tonTimer2.Q THEN
			sReactorError												:= gsRepressurizationError;
		END_IF
		
	4:
		bTimer1															:= TRUE;
		IF R_S.all_clamps_retracted THEN																					// 2.a.iv
			bTimer1														:= FALSE;
			R_S.open_repres_valves										:= TRUE;
			i4Step														:= i4Step + 2;
		ELSIF tonTimer1.Q THEN
			bTimer1														:= FALSE;
			sReactorError												:= gsDoorClampsExtendedError;
			sMessage													:= gsProcessCannotRun;
		END_IF
		
	5:
		bTimer1															:= TRUE;											// 4
		IF R_S.dead_air_valve_clear THEN
			bTimer1														:= FALSE;
			i4Step														:= i4Step + 1;
		ELSIF tonTimer1.Q THEN
			bTimer1														:= FALSE;
			sReactorError												:= gsDeadAirValveError;
		END_IF

	6:
		IF R_S.average_reactor_pressure	>= m01.SP_repres_pres_highlimit THEN		
			i4Step														:= 99;
		END_IF			
			
	7:
		bTimer1															:= TRUE;
		IF tonTimer1.Q THEN
			R_S.open_repres_valves										:= FALSE;
			i4Step														:= 99;
		END_IF
	
	80:																														// Manual process closing
		Cycle_Stage														:= 'repressurization.stopping';
		R_S.co2_sensors_off												:= TRUE;
		R_S.close_repres_valves											:= TRUE;
		U.drainage_on													:= FALSE;
		rTime1															:= _STOPPING_TIME;
		i4Step															:= i4Step + 1;
		
	81:
		bTimer1															:= TRUE;
		IF tonTimer1.Q THEN
			bTimer1														:= FALSE;
			i4Step														:= 99;
		END_IF
		
	90:																														// Automatic process stopping
		Cycle_Stage														:= 'repressurization.stopping';
		R_S.co2_sensors_off												:= TRUE;
		R_S.close_repres_valves											:= TRUE;
		U.drainage_on													:= FALSE;
		rTime1															:= _STOPPING_TIME;
		i4Step															:= i4Step + 1;
		
	91:
		bTimer1															:= TRUE;
		IF tonTimer1.Q THEN
			bTimer1														:= FALSE;
			i4Step														:= 99;
		END_IF
		
	98:																														// Utility error hold - cleared by P_M01
		i4Step															:= 98;
		
	99:
		bRepressurizationDone											:= TRUE;
		Current_Step													:= 0;
		i4Step															:= 0;
	
END_CASE

IF i4Step > 0 AND i4Step < 80 THEN
	IF bMultiProcess THEN
		IF U.safe_shutdown_error_1 <> '' AND giSafeShutdown1RS = 0 THEN
			sSafeShutdownError1											:= U.safe_shutdown_error_1;
			giSafeShutdown1RS											:= RS_Number;
		ELSIF U.safe_shutdown_error_2 <> '' AND giSafeShutdown23RS = 0 THEN
			sSafeShutdownError2											:= U.safe_shutdown_error_2;
			giSafeShutdown23RS											:= RS_Number;
		ELSIF (giEvacuationErrorRS + giDesorptionErrorRS + giSafeShutdown1RS + giSafeShutdown23RS) > 0 THEN
			Cancel_Reactor_Set											:= TRUE;
		ELSIF U.os_air_unsafe_temp THEN
			Stop_Reactor_Set											:= TRUE;
		END_IF
	END_IF
	iStep																:= i4Step;
	Current_Step														:= iStep;
	A_Check_Process();
	i4Step																:= iStep;
END_IF
END_ACTION

ACTION A4_Repressurization_Test_Auto:
// Phase 0 - FB_Reactor_Set.A4_Repressurization_Test
// Rev 1.0 - June 3, 2024

CASE i4Step OF
	
	0:	;
		
	1:
		Cycle_Stage														:= 'repressurization.initialize';					// 2.a.i and 4.i
		rTime1														:= _VALVE_TIME;
		Steam_Service_Req											:= TRUE;
		IF Steam_Service_Assigned THEN 
			i4Step														:= i4Step + 1;
		END_IF
			
	2:
		bTimer1															:= TRUE;
		IF sita_bits[4].1 THEN 
			bTimer1														:= FALSE;
			i4Step														:= 90;
		ELSIF tonTimer1.Q AND  sita_bits[4].2 THEN 
			bTimer1														:= FALSE;
			sReactorError												:= 'Repress Error';
			sMessage													:= 'Auto Test';
		END_IF
		
	
	80:																														// Manual process closing
		Cycle_Stage														:= 'repressurization.stopping';
		rTime1															:= _STOPPING_TIME;
		i4Step															:= i4Step + 1;
		
	81:
		bTimer1															:= TRUE;
		IF tonTimer1.Q THEN
			bTimer1														:= FALSE;
			i4Step														:= 99;
		END_IF
		
	90:																														// Automatic process stopping
		Cycle_Stage														:= 'repressurization.stopping';
		R_S.co2_sensors_off												:= TRUE;
		R_S.close_repres_valves											:= TRUE;
		U.drainage_on													:= FALSE;
		rTime1															:= _STOPPING_TIME;
		i4Step															:= i4Step + 1;
		
